LIN {X 0,Y 249.079,Z 319.46,A -85,B 0,C 180,E1 -18873.163,E2 -18873.163} C_VEL
LIN {X 0,Y 249.068,Z 319.458,A -85,B 0,C 180,E1 -18876.731,E2 -18876.731} C_VEL
LIN {X 0,Y 249.086,Z 319.447,A -85,B 0,C 180,E1 -18880.209,E2 -18880.209} C_VEL
LIN {X 0,Y 249.185,Z 319.436,A -85,B 0,C 180,E1 -18883.618,E2 -18883.618} C_VEL
LIN {X 0,Y 249.22,Z 319.439,A -85,B 0,C 180,E1 -18886.961,E2 -18886.961} C_VEL
LIN {X 0,Y 249.392,Z 319.411,A -85,B 0,C 180,E1 -18890.522,E2 -18890.522} C_VEL
LIN {X 0,Y 249.437,Z 319.395,A -85,B 0,C 180,E1 -18893.529,E2 -18893.529} C_VEL
LIN {X 0,Y 249.681,Z 319.382,A -85,B 0,C 180,E1 -18898.387,E2 -18898.387} C_VEL
LIN {X 0,Y 249.681,Z 319.38,A -85,B 0,C 180,E1 -18901.613,E2 -18901.613} C_VEL
LIN {X 0,Y 249.441,Z 319.394,A -85,B 0,C 180,E1 -18906.7,E2 -18906.7} C_VEL
LIN {X 0,Y 249.351,Z 319.418,A -85,B 0,C 180,E1 -18909.736,E2 -18909.736} C_VEL
LIN {X 0,Y 249.179,Z 319.442,A -85,B 0,C 180,E1 -18914.705,E2 -18914.705} C_VEL
LIN {X 0,Y 249.11,Z 319.452,A -85,B 0,C 180,E1 -18918.079,E2 -18918.079} C_VEL
LIN {X 0,Y 249.088,Z 319.452,A -85,B 0,C 180,E1 -18921.518,E2 -18921.518} C_VEL
LIN {X 0,Y 249.123,Z 319.451,A -85,B 0,C 180,E1 -18925.474,E2 -18925.474} C_VEL
LIN {X 0,Y 249.089,Z 319.453,A -85,B 0,C 180,E1 -18928.992,E2 -18928.992} C_VEL
LIN {X 0,Y 249.037,Z 319.46,A -85,B 0,C 180,E1 -18932.425,E2 -18932.425} C_VEL
LIN {X 0,Y 249.035,Z 319.459,A -85,B 0,C 180,E1 -18936.344,E2 -18936.344} C_VEL
LIN {X 0,Y 249.013,Z 319.458,A -85,B 0,C 180,E1 -18940.476,E2 -18940.476} C_VEL
LIN {X 0,Y 249.017,Z 319.462,A -85,B 0,C 180,E1 -18942.792,E2 -18942.792} C_VEL
LIN {X 0,Y 249.014,Z 319.464,A -85,B 0,C 180,E1 -18947.36,E2 -18947.36} C_VEL
LIN {X 0,Y 249.031,Z 319.463,A -85,B 0,C 180,E1 -18951.618,E2 -18951.618} C_VEL
LIN {X 0,Y 249.048,Z 319.46,A -85,B 0,C 180,E1 -18955.638,E2 -18955.638} C_VEL
LIN {X 0,Y 249.052,Z 319.46,A -85,B 0,C 180,E1 -18959.471,E2 -18959.471} C_VEL
LIN {X 0,Y 249.076,Z 319.457,A -85,B 0,C 180,E1 -18963.16,E2 -18963.16} C_VEL
LIN {X 0,Y 249.088,Z 319.457,A -85,B 0,C 180,E1 -18966.731,E2 -18966.731} C_VEL
LIN {X 0,Y 249.134,Z 319.449,A -85,B 0,C 180,E1 -18970.211,E2 -18970.211} C_VEL
LIN {X 0,Y 249.245,Z 319.438,A -85,B 0,C 180,E1 -18973.62,E2 -18973.62} C_VEL
LIN {X 0,Y 249.223,Z 319.441,A -85,B 0,C 180,E1 -18975.732,E2 -18975.732} C_VEL
LIN {X 0,Y 250.259,Z 322.319,A -85,B 0,C 180,E1 -18975.945,E2 -18975.945} C_VEL
LIN {X 0,Y 254.771,Z 333.047,A -85,B 0,C 180,E1 -18976.726,E2 -18976.726} C_VEL
LIN {X 0,Y 260.864,Z 350.4,A -85,B 0,C 180,E1 -18977.82,E2 -18977.82} C_VEL
LIN {X 0,Y 261.655,Z 353.279,A -85,B 0,C 180,E1 -18977.976,E2 -18977.976} C_VEL
LIN {X 0,Y 259.286,Z 425.995,A -85,B 0,C 180,E1 -18979.952,E2 -18979.952} C_VEL
LIN {X 0,Y 258.532,Z 439.131,A -85,B 0,C 180,E1 -18980.611,E2 -18980.611} C_VEL
LIN {X 0,Y 257.521,Z 451.819,A -85,B 0,C 180,E1 -18981.563,E2 -18981.563} C_VEL
LIN {X 0,Y 256.275,Z 463.159,A -85,B 0,C 180,E1 -18982.711,E2 -18982.711} C_VEL
LIN {X 0,Y 254.783,Z 475.126,A -85,B 0,C 180,E1 -18984.307,E2 -18984.307} C_VEL
LIN {X 0,Y 253.083,Z 486.09,A -85,B 0,C 180,E1 -18986.156,E2 -18986.156} C_VEL
LIN {X 0,Y 251.687,Z 494.8,A -85,B 0,C 180,E1 -18987.997,E2 -18987.997} C_VEL
LIN {X 0,Y 250.106,Z 503.926,A -85,B 0,C 180,E1 -18990.4,E2 -18990.4} C_VEL
LIN {X 0,Y 248.944,Z 511.268,A -85,B 0,C 180,E1 -18992.829,E2 -18992.829} C_VEL
LIN {X 0,Y 248.22,Z 516.233,A -85,B 0,C 180,E1 -18994.87,E2 -18994.87} C_VEL
LIN {X 0,Y 247.608,Z 521.055,A -85,B 0,C 180,E1 -18997.335,E2 -18997.335} C_VEL
LIN {X 0,Y 247.108,Z 524.766,A -85,B 0,C 180,E1 -18999.823,E2 -18999.823} C_VEL
LIN {X 0,Y 246.862,Z 526.683,A -85,B 0,C 180,E1 -19001.493,E2 -19001.493} C_VEL
LIN {X 0,Y 246.746,Z 528.928,A -85,B 0,C 180,E1 -19004.441,E2 -19004.441} C_VEL
LIN {X 0,Y 246.751,Z 529.759,A -85,B 0,C 180,E1 -19006.545,E2 -19006.545} C_VEL
LIN {X 0,Y 246.908,Z 529.939,A -85,B 0,C 180,E1 -19008.244,E2 -19008.244} C_VEL
LIN {X 0,Y 247.271,Z 529.588,A -85,B 0,C 180,E1 -19010.293,E2 -19010.293} C_VEL
LIN {X 0,Y 248.086,Z 527.931,A -85,B 0,C 180,E1 -19013.363,E2 -19013.363} C_VEL
LIN {X 0,Y 248.951,Z 525.994,A -85,B 0,C 180,E1 -19015.395,E2 -19015.395} C_VEL
LIN {X 0,Y 250.625,Z 521.798,A -85,B 0,C 180,E1 -19018.468,E2 -19018.468} C_VEL
LIN {X 0,Y 252.431,Z 516.954,A -85,B 0,C 180,E1 -19020.998,E2 -19020.998} C_VEL
LIN {X 0,Y 254.728,Z 510.734,A -85,B 0,C 180,E1 -19023.488,E2 -19023.488} C_VEL
LIN {X 0,Y 257.367,Z 502.891,A -85,B 0,C 180,E1 -19025.949,E2 -19025.949} C_VEL
LIN {X 0,Y 259.932,Z 494.763,A -85,B 0,C 180,E1 -19027.956,E2 -19027.956} C_VEL
LIN {X 0,Y 262.477,Z 485.797,A -85,B 0,C 180,E1 -19029.739,E2 -19029.739} C_VEL
LIN {X 0,Y 265.25,Z 474.762,A -85,B 0,C 180,E1 -19031.479,E2 -19031.479} C_VEL
LIN {X 0,Y 267.697,Z 463.298,A -85,B 0,C 180,E1 -19032.887,E2 -19032.887} C_VEL
LIN {X 0,Y 269.763,Z 450.842,A -85,B 0,C 180,E1 -19034.045,E2 -19034.045} C_VEL
LIN {X 0,Y 271.36,Z 438.352,A -85,B 0,C 180,E1 -19034.884,E2 -19034.884} C_VEL
LIN {X 0,Y 272.421,Z 425.844,A -85,B 0,C 180,E1 -19035.444,E2 -19035.444} C_VEL
LIN {X 0,Y 274.997,Z 366.968,A -85,B 0,C 180,E1 -19036.992,E2 -19036.992} C_VEL
LIN {X 0,Y 268.888,Z 353.819,A -85,B 0,C 180,E1 -19038.45,E2 -19038.45} C_VEL
LIN {X 0,Y 262.221,Z 341.314,A -85,B 0,C 180,E1 -19040.095,E2 -19040.095} C_VEL
LIN {X 0,Y 254.553,Z 328.6,A -85,B 0,C 180,E1 -19042.099,E2 -19042.099} C_VEL
LIN {X 0,Y 251.261,Z 323.754,A -85,B 0,C 180,E1 -19042.995,E2 -19042.995} C_VEL
LIN {X 0,Y 249.526,Z 321.295,A -85,B 0,C 180,E1 -19043.479,E2 -19043.479} C_VEL
LIN {X 0,Y 249.129,Z 320.072,A -85,B 0,C 180,E1 -19043.672,E2 -19043.672} C_VEL
LIN {X 0,Y 249.026,Z 319.443,A -85,B 0,C 180,E1 -19044.008,E2 -19044.008} C_VEL
LIN {X 0,Y 249.021,Z 319.463,A -85,B 0,C 180,E1 -19047.846,E2 -19047.846} C_VEL
LIN {X 0,Y 249.036,Z 319.458,A -85,B 0,C 180,E1 -19051.331,E2 -19051.331} C_VEL
LIN {X 0,Y 249.089,Z 319.449,A -85,B 0,C 180,E1 -19054.962,E2 -19054.962} C_VEL
LIN {X 0,Y 249.081,Z 319.448,A -85,B 0,C 180,E1 -19058.602,E2 -19058.602} C_VEL
LIN {X 0,Y 249.23,Z 319.427,A -85,B 0,C 180,E1 -19063.621,E2 -19063.621} C_VEL
LIN {X 0,Y 249.232,Z 319.427,A -85,B 0,C 180,E1 -19068.616,E2 -19068.616} C_VEL
LIN {X 0,Y 249.423,Z 319.406,A -85,B 0,C 180,E1 -19071.901,E2 -19071.901} C_VEL
LIN {X 0,Y 249.418,Z 319.409,A -85,B 0,C 180,E1 -19076.77,E2 -19076.77} C_VEL
LIN {X 0,Y 249.715,Z 319.375,A -85,B 0,C 180,E1 -19080,E2 -19080} C_VEL
LIN {X 0,Y 249.421,Z 319.397,A -85,B 0,C 180,E1 -19083.231,E2 -19083.231} C_VEL
LIN {X 0,Y 249.447,Z 319.398,A -85,B 0,C 180,E1 -19087.739,E2 -19087.739} C_VEL
LIN {X 0,Y 248.791,Z 319.482,A -85,B 0,C 180,E1 -19089.084,E2 -19089.084} C_VEL
LIN {X 0,Y 245.807,Z 319.865,A -85,B 0,C 180,E1 -19091.272,E2 -19091.272} C_VEL
LIN {X 0,Y 243.266,Z 320.171,A -85,B 0,C 180,E1 -19093.055,E2 -19093.055} C_VEL
LIN {X 0,Y 242.208,Z 320.299,A -85,B 0,C 180,E1 -19094.443,E2 -19094.443} C_VEL
LIN {X 0,Y 242.142,Z 320.311,A -85,B 0,C 180,E1 -19094.913,E2 -19094.913} C_VEL
LIN {X 0,Y 242.062,Z 320.318,A -85,B 0,C 180,E1 -19098.625,E2 -19098.625} C_VEL
LIN {X 0,Y 242.002,Z 320.336,A -85,B 0,C 180,E1 -19102.181,E2 -19102.181} C_VEL
LIN {X 0,Y 242.056,Z 320.334,A -85,B 0,C 180,E1 -19105.84,E2 -19105.84} C_VEL
LIN {X 0,Y 242.021,Z 320.335,A -85,B 0,C 180,E1 -19109.582,E2 -19109.582} C_VEL
LIN {X 0,Y 241.982,Z 320.341,A -85,B 0,C 180,E1 -19113.493,E2 -19113.493} C_VEL
LIN {X 0,Y 242.005,Z 320.345,A -85,B 0,C 180,E1 -19117.58,E2 -19117.58} C_VEL
LIN {X 0,Y 241.962,Z 320.342,A -85,B 0,C 180,E1 -19121.918,E2 -19121.918} C_VEL
LIN {X 0,Y 241.956,Z 320.354,A -85,B 0,C 180,E1 -19123.861,E2 -19123.861} C_VEL
LIN {X 0,Y 244.234,Z 327.54,A -85,B 0,C 180,E1 -19127.815,E2 -19127.815} C_VEL
LIN {X 0,Y 245.915,Z 333.614,A -85,B 0,C 180,E1 -19130.733,E2 -19130.733} C_VEL
LIN {X 0,Y 248.478,Z 338.048,A -85,B 0,C 180,E1 -19131.493,E2 -19131.493} C_VEL
LIN {X 0,Y 254.393,Z 348.559,A -85,B 0,C 180,E1 -19133.168,E2 -19133.168} C_VEL
LIN {X 0,Y 260.731,Z 361.176,A -85,B 0,C 180,E1 -19134.877,E2 -19134.877} C_VEL
LIN {X 0,Y 265.439,Z 371.761,A -85,B 0,C 180,E1 -19136.103,E2 -19136.103} C_VEL
LIN {X 0,Y 268.42,Z 390.693,A -85,B 0,C 180,E1 -19137.259,E2 -19137.259} C_VEL
LIN {X 0,Y 265.995,Z 443.364,A -85,B 0,C 180,E1 -19138.684,E2 -19138.684} C_VEL
LIN {X 0,Y 264.584,Z 457.091,A -85,B 0,C 180,E1 -19139.33,E2 -19139.33} C_VEL
LIN {X 0,Y 262.579,Z 469.788,A -85,B 0,C 180,E1 -19140.213,E2 -19140.213} C_VEL
LIN {X 0,Y 260.163,Z 481.585,A -85,B 0,C 180,E1 -19141.351,E2 -19141.351} C_VEL
LIN {X 0,Y 257.684,Z 491.661,A -85,B 0,C 180,E1 -19142.6,E2 -19142.6} C_VEL
LIN {X 0,Y 254.822,Z 502.14,A -85,B 0,C 180,E1 -19144.257,E2 -19144.257} C_VEL
LIN {X 0,Y 251.917,Z 511.618,A -85,B 0,C 180,E1 -19146.142,E2 -19146.142} C_VEL
LIN {X 0,Y 248.731,Z 520.781,A -85,B 0,C 180,E1 -19148.452,E2 -19148.452} C_VEL
LIN {X 0,Y 246.35,Z 528.171,A -85,B 0,C 180,E1 -19150.851,E2 -19150.851} C_VEL
LIN {X 0,Y 244.26,Z 534.136,A -85,B 0,C 180,E1 -19153.281,E2 -19153.281} C_VEL
LIN {X 0,Y 242.422,Z 538.878,A -85,B 0,C 180,E1 -19155.737,E2 -19155.737} C_VEL
LIN {X 0,Y 241.211,Z 542.533,A -85,B 0,C 180,E1 -19158.234,E2 -19158.234} C_VEL
LIN {X 0,Y 240.639,Z 544.439,A -85,B 0,C 180,E1 -19159.91,E2 -19159.91} C_VEL
LIN {X 0,Y 240.214,Z 545.898,A -85,B 0,C 180,E1 -19161.591,E2 -19161.591} C_VEL
LIN {X 0,Y 239.841,Z 547.621,A -85,B 0,C 180,E1 -19164.959,E2 -19164.959} C_VEL
LIN {X 0,Y 239.82,Z 547.911,A -85,B 0,C 180,E1 -19166.642,E2 -19166.642} C_VEL
LIN {X 0,Y 239.903,Z 547.793,A -85,B 0,C 180,E1 -19168.324,E2 -19168.324} C_VEL
LIN {X 0,Y 239.958,Z 547.253,A -85,B 0,C 180,E1 -19170.003,E2 -19170.003} C_VEL
LIN {X 0,Y 239.953,Z 546.315,A -85,B 0,C 180,E1 -19171.681,E2 -19171.681} C_VEL
LIN {X 0,Y 239.892,Z 544.97,A -85,B 0,C 180,E1 -19173.362,E2 -19173.362} C_VEL
LIN {X 0,Y 239.922,Z 542.099,A -85,B 0,C 180,E1 -19175.886,E2 -19175.886} C_VEL
LIN {X 0,Y 240.201,Z 538.173,A -85,B 0,C 180,E1 -19178.415,E2 -19178.415} C_VEL
LIN {X 0,Y 240.827,Z 532.102,A -85,B 0,C 180,E1 -19181.363,E2 -19181.363} C_VEL
LIN {X 0,Y 241.786,Z 525.416,A -85,B 0,C 180,E1 -19183.877,E2 -19183.877} C_VEL
LIN {X 0,Y 243.16,Z 517.097,A -85,B 0,C 180,E1 -19186.37,E2 -19186.37} C_VEL
LIN {X 0,Y 244.587,Z 508.167,A -85,B 0,C 180,E1 -19188.516,E2 -19188.516} C_VEL
LIN {X 0,Y 246.257,Z 497.98,A -85,B 0,C 180,E1 -19190.466,E2 -19190.466} C_VEL
LIN {X 0,Y 247.77,Z 487.482,A -85,B 0,C 180,E1 -19192.078,E2 -19192.078} C_VEL
LIN {X 0,Y 249.502,Z 476.011,A -85,B 0,C 180,E1 -19193.448,E2 -19193.448} C_VEL
LIN {X 0,Y 250.861,Z 464.137,A -85,B 0,C 180,E1 -19194.52,E2 -19194.52} C_VEL
LIN {X 0,Y 251.995,Z 451.358,A -85,B 0,C 180,E1 -19195.338,E2 -19195.338} C_VEL
LIN {X 0,Y 252.7,Z 438.181,A -85,B 0,C 180,E1 -19195.87,E2 -19195.87} C_VEL
LIN {X 0,Y 254.188,Z 385.832,A -85,B 0,C 180,E1 -19197.324,E2 -19197.324} C_VEL
LIN {X 0,Y 249.433,Z 347.285,A -85,B 0,C 180,E1 -19198.962,E2 -19198.962} C_VEL
LIN {X 0,Y 245.183,Z 335.103,A -85,B 0,C 180,E1 -19199.805,E2 -19199.805} C_VEL
LIN {X 0,Y 242.879,Z 324.284,A -85,B 0,C 180,E1 -19203.853,E2 -19203.853} C_VEL
LIN {X 0,Y 242.016,Z 320.338,A -85,B 0,C 180,E1 -19205.445,E2 -19205.445} C_VEL
LIN {X 0,Y 241.963,Z 320.345,A -85,B 0,C 180,E1 -19209.72,E2 -19209.72} C_VEL
LIN {X 0,Y 241.926,Z 320.349,A -85,B 0,C 180,E1 -19214.206,E2 -19214.206} C_VEL
LIN {X 0,Y 241.941,Z 320.346,A -85,B 0,C 180,E1 -19218.078,E2 -19218.078} C_VEL
LIN {X 0,Y 241.994,Z 320.338,A -85,B 0,C 180,E1 -19222.418,E2 -19222.418} C_VEL
LIN {X 0,Y 241.988,Z 320.337,A -85,B 0,C 180,E1 -19226.508,E2 -19226.508} C_VEL
LIN {X 0,Y 242.045,Z 320.329,A -85,B 0,C 180,E1 -19230.588,E2 -19230.588} C_VEL
LIN {X 0,Y 242.076,Z 320.329,A -85,B 0,C 180,E1 -19234.184,E2 -19234.184} C_VEL
LIN {X 0,Y 242.031,Z 320.333,A -85,B 0,C 180,E1 -19238.316,E2 -19238.316} C_VEL
LIN {X 0,Y 242.124,Z 320.312,A -85,B 0,C 180,E1 -19243.316,E2 -19243.316} C_VEL
LIN {X 0,Y 242.186,Z 320.314,A -85,B 0,C 180,E1 -19248.279,E2 -19248.279} C_VEL
LIN {X 0,Y 242.38,Z 320.279,A -85,B 0,C 180,E1 -19251.664,E2 -19251.664} C_VEL
LIN {X 0,Y 242.249,Z 320.295,A -85,B 0,C 180,E1 -19255.007,E2 -19255.007} C_VEL
LIN {X 0,Y 242.642,Z 320.259,A -85,B 0,C 180,E1 -19258.34,E2 -19258.34} C_VEL
LIN {X 0,Y 242.642,Z 320.257,A -85,B 0,C 180,E1 -19261.659,E2 -19261.659} C_VEL
LIN {X 0,Y 242.423,Z 320.268,A -85,B 0,C 180,E1 -19266.672,E2 -19266.672} C_VEL
LIN {X 0,Y 242.275,Z 320.3,A -85,B 0,C 180,E1 -19270.023,E2 -19270.023} C_VEL
LIN {X 0,Y 242.134,Z 320.317,A -85,B 0,C 180,E1 -19275.143,E2 -19275.143} C_VEL
LIN {X 0,Y 242.049,Z 320.335,A -85,B 0,C 180,E1 -19278.626,E2 -19278.626} C_VEL
LIN {X 0,Y 242.011,Z 320.333,A -85,B 0,C 180,E1 -19282.18,E2 -19282.18} C_VEL
LIN {X 0,Y 242.074,Z 320.328,A -85,B 0,C 180,E1 -19285.837,E2 -19285.837} C_VEL
LIN {X 0,Y 242.037,Z 320.331,A -85,B 0,C 180,E1 -19289.579,E2 -19289.579} C_VEL
LIN {X 0,Y 241.987,Z 320.337,A -85,B 0,C 180,E1 -19293.491,E2 -19293.491} C_VEL
LIN {X 0,Y 241.993,Z 320.339,A -85,B 0,C 180,E1 -19297.581,E2 -19297.581} C_VEL
LIN {X 0,Y 241.945,Z 320.344,A -85,B 0,C 180,E1 -19301.92,E2 -19301.92} C_VEL
LIN {X 0,Y 241.932,Z 320.344,A -85,B 0,C 180,E1 -19306.571,E2 -19306.571} C_VEL
LIN {X 0,Y 241.961,Z 320.341,A -85,B 0,C 180,E1 -19310.279,E2 -19310.279} C_VEL
LIN {X 0,Y 241.993,Z 320.338,A -85,B 0,C 180,E1 -19314.488,E2 -19314.488} C_VEL
LIN {X 0,Y 241.977,Z 320.341,A -85,B 0,C 180,E1 -19318.478,E2 -19318.478} C_VEL
LIN {X 0,Y 242.007,Z 320.339,A -85,B 0,C 180,E1 -19322.31,E2 -19322.31} C_VEL
LIN {X 0,Y 242.064,Z 320.333,A -85,B 0,C 180,E1 -19326.014,E2 -19326.014} C_VEL
LIN {X 0,Y 242.064,Z 320.329,A -85,B 0,C 180,E1 -19329.608,E2 -19329.608} C_VEL
LIN {X 0,Y 242.166,Z 320.32,A -85,B 0,C 180,E1 -19333.276,E2 -19333.276} C_VEL
LIN {X 0,Y 242.169,Z 320.318,A -85,B 0,C 180,E1 -19334.988,E2 -19334.988} C_VEL
LIN {X 0,Y 243.233,Z 323.279,A -85,B 0,C 180,E1 -19335.234,E2 -19335.234} C_VEL
LIN {X 0,Y 247.549,Z 332.958,A -85,B 0,C 180,E1 -19336,E2 -19336} C_VEL
LIN {X 0,Y 254.442,Z 352.277,A -85,B 0,C 180,E1 -19337.282,E2 -19337.282} C_VEL
LIN {X 0,Y 255.026,Z 354.157,A -85,B 0,C 180,E1 -19337.394,E2 -19337.394} C_VEL
LIN {X 0,Y 252.608,Z 426.79,A -85,B 0,C 180,E1 -19339.427,E2 -19339.427} C_VEL
LIN {X 0,Y 251.761,Z 440.555,A -85,B 0,C 180,E1 -19340.153,E2 -19340.153} C_VEL
LIN {X 0,Y 250.737,Z 452.917,A -85,B 0,C 180,E1 -19341.13,E2 -19341.13} C_VEL
LIN {X 0,Y 249.425,Z 464.032,A -85,B 0,C 180,E1 -19342.306,E2 -19342.306} C_VEL
LIN {X 0,Y 248.065,Z 474.734,A -85,B 0,C 180,E1 -19343.767,E2 -19343.767} C_VEL
LIN {X 0,Y 246.256,Z 486.013,A -85,B 0,C 180,E1 -19345.701,E2 -19345.701} C_VEL
LIN {X 0,Y 244.832,Z 494.536,A -85,B 0,C 180,E1 -19347.53,E2 -19347.53} C_VEL
LIN {X 0,Y 243.197,Z 503.765,A -85,B 0,C 180,E1 -19349.998,E2 -19349.998} C_VEL
LIN {X 0,Y 241.966,Z 511.183,A -85,B 0,C 180,E1 -19352.495,E2 -19352.495} C_VEL
LIN {X 0,Y 241.093,Z 517.128,A -85,B 0,C 180,E1 -19355.014,E2 -19355.014} C_VEL
LIN {X 0,Y 240.473,Z 521.82,A -85,B 0,C 180,E1 -19357.554,E2 -19357.554} C_VEL
LIN {X 0,Y 239.953,Z 525.411,A -85,B 0,C 180,E1 -19360.119,E2 -19360.119} C_VEL
LIN {X 0,Y 239.75,Z 527.213,A -85,B 0,C 180,E1 -19361.838,E2 -19361.838} C_VEL
LIN {X 0,Y 239.655,Z 529.203,A -85,B 0,C 180,E1 -19364.594,E2 -19364.594} C_VEL
LIN {X 0,Y 239.684,Z 530.09,A -85,B 0,C 180,E1 -19367.048,E2 -19367.048} C_VEL
LIN {X 0,Y 239.893,Z 530.183,A -85,B 0,C 180,E1 -19368.797,E2 -19368.797} C_VEL
LIN {X 0,Y 240.24,Z 529.86,A -85,B 0,C 180,E1 -19370.589,E2 -19370.589} C_VEL
LIN {X 0,Y 240.656,Z 529.148,A -85,B 0,C 180,E1 -19372.309,E2 -19372.309} C_VEL
LIN {X 0,Y 241.257,Z 527.942,A -85,B 0,C 180,E1 -19374.066,E2 -19374.066} C_VEL
LIN {X 0,Y 242.475,Z 525.304,A -85,B 0,C 180,E1 -19376.692,E2 -19376.692} C_VEL
LIN {X 0,Y 244.055,Z 521.552,A -85,B 0,C 180,E1 -19379.308,E2 -19379.308} C_VEL
LIN {X 0,Y 246.032,Z 516.566,A -85,B 0,C 180,E1 -19381.898,E2 -19381.898} C_VEL
LIN {X 0,Y 248.51,Z 510.192,A -85,B 0,C 180,E1 -19384.441,E2 -19384.441} C_VEL
LIN {X 0,Y 251.388,Z 502.122,A -85,B 0,C 180,E1 -19386.943,E2 -19386.943} C_VEL
LIN {X 0,Y 254.274,Z 493.012,A -85,B 0,C 180,E1 -19389.158,E2 -19389.158} C_VEL
LIN {X 0,Y 257.105,Z 483.439,A -85,B 0,C 180,E1 -19390.995,E2 -19390.995} C_VEL
LIN {X 0,Y 259.708,Z 473.148,A -85,B 0,C 180,E1 -19392.569,E2 -19392.569} C_VEL
LIN {X 0,Y 262.245,Z 461.061,A -85,B 0,C 180,E1 -19394.002,E2 -19394.002} C_VEL
LIN {X 0,Y 264.216,Z 449.064,A -85,B 0,C 180,E1 -19395.086,E2 -19395.086} C_VEL
LIN {X 0,Y 265.774,Z 436.705,A -85,B 0,C 180,E1 -19395.877,E2 -19395.877} C_VEL
LIN {X 0,Y 266.835,Z 424.087,A -85,B 0,C 180,E1 -19396.394,E2 -19396.394} C_VEL
LIN {X 0,Y 269.338,Z 369.122,A -85,B 0,C 180,E1 -19397.852,E2 -19397.852} C_VEL
LIN {X 0,Y 263.234,Z 356.083,A -85,B 0,C 180,E1 -19399.377,E2 -19399.377} C_VEL
LIN {X 0,Y 255.57,Z 342.012,A -85,B 0,C 180,E1 -19401.376,E2 -19401.376} C_VEL
LIN {X 0,Y 249.809,Z 332.638,A -85,B 0,C 180,E1 -19402.962,E2 -19402.962} C_VEL
LIN {X 0,Y 247.435,Z 329.138,A -85,B 0,C 180,E1 -19403.636,E2 -19403.636} C_VEL
LIN {X 0,Y 245.35,Z 326.004,A -85,B 0,C 180,E1 -19404.247,E2 -19404.247} C_VEL
LIN {X 0,Y 244.417,Z 324.846,A -85,B 0,C 180,E1 -19404.516,E2 -19404.516} C_VEL
LIN {X 0,Y 242.517,Z 322.265,A -85,B 0,C 180,E1 -19405.087,E2 -19405.087} C_VEL
LIN {X 0,Y 242.018,Z 320.518,A -85,B 0,C 180,E1 -19405.321,E2 -19405.321} C_VEL
LIN {X 0,Y 241.94,Z 320.342,A -85,B 0,C 180,E1 -19408.475,E2 -19408.475} C_VEL
LIN {X 0,Y 241.955,Z 320.34,A -85,B 0,C 180,E1 -19412.307,E2 -19412.307} C_VEL
LIN {X 0,Y 242.013,Z 320.332,A -85,B 0,C 180,E1 -19416.012,E2 -19416.012} C_VEL
LIN {X 0,Y 242.023,Z 320.326,A -85,B 0,C 180,E1 -19419.607,E2 -19419.607} C_VEL
LIN {X 0,Y 242.151,Z 320.308,A -85,B 0,C 180,E1 -19423.278,E2 -19423.278} C_VEL
LIN {X 0,Y 242.168,Z 320.305,A -85,B 0,C 180,E1 -19428.279,E2 -19428.279} C_VEL
LIN {X 0,Y 242.373,Z 320.286,A -85,B 0,C 180,E1 -19431.664,E2 -19431.664} C_VEL
LIN {X 0,Y 242.233,Z 320.31,A -85,B 0,C 180,E1 -19435.007,E2 -19435.007} C_VEL
LIN {X 0,Y 242.622,Z 320.246,A -85,B 0,C 180,E1 -19438.34,E2 -19438.34} C_VEL
LIN {X 0,Y 242.623,Z 320.258,A -85,B 0,C 180,E1 -19441.66,E2 -19441.66} C_VEL
LIN {X 0,Y 242.394,Z 320.276,A -85,B 0,C 180,E1 -19447.745,E2 -19447.745} C_VEL
LIN {X 0,Y 242.302,Z 320.295,A -85,B 0,C 180,E1 -19450.023,E2 -19450.023} C_VEL
LIN {X 0,Y 242.142,Z 320.311,A -85,B 0,C 180,E1 -19454.913,E2 -19454.913} C_VEL
LIN {X 0,Y 241.521,Z 320.402,A -85,B 0,C 180,E1 -19456.3,E2 -19456.3} C_VEL
LIN {X 0,Y 238.655,Z 320.771,A -85,B 0,C 180,E1 -19458.561,E2 -19458.561} C_VEL
LIN {X 0,Y 236.167,Z 321.077,A -85,B 0,C 180,E1 -19460.403,E2 -19460.403} C_VEL
LIN {X 0,Y 235.069,Z 321.203,A -85,B 0,C 180,E1 -19461.834,E2 -19461.834} C_VEL
LIN {X 0,Y 234.965,Z 321.21,A -85,B 0,C 180,E1 -19462.319,E2 -19462.319} C_VEL
LIN {X 0,Y 234.96,Z 321.213,A -85,B 0,C 180,E1 -19466.659,E2 -19466.659} C_VEL
LIN {X 0,Y 234.923,Z 321.223,A -85,B 0,C 180,E1 -19470.569,E2 -19470.569} C_VEL
LIN {X 0,Y 234.952,Z 321.219,A -85,B 0,C 180,E1 -19474.635,E2 -19474.635} C_VEL
LIN {X 0,Y 234.959,Z 321.214,A -85,B 0,C 180,E1 -19478.954,E2 -19478.954} C_VEL
LIN {X 0,Y 234.927,Z 321.303,A -85,B 0,C 180,E1 -19482.328,E2 -19482.328} C_VEL
LIN {X 0,Y 237.543,Z 329.57,A -85,B 0,C 180,E1 -19487.123,E2 -19487.123} C_VEL
LIN {X 0,Y 238.558,Z 333.073,A -85,B 0,C 180,E1 -19488.923,E2 -19488.923} C_VEL
LIN {X 0,Y 241.281,Z 337.753,A -85,B 0,C 180,E1 -19489.806,E2 -19489.806} C_VEL
LIN {X 0,Y 247.872,Z 349.115,A -85,B 0,C 180,E1 -19491.802,E2 -19491.802} C_VEL
LIN {X 0,Y 254.514,Z 362.104,A -85,B 0,C 180,E1 -19493.704,E2 -19493.704} C_VEL
LIN {X 0,Y 260.214,Z 374.792,A -85,B 0,C 180,E1 -19495.271,E2 -19495.271} C_VEL
LIN {X 0,Y 262.808,Z 391.644,A -85,B 0,C 180,E1 -19496.334,E2 -19496.334} C_VEL
LIN {X 0,Y 260.27,Z 443.79,A -85,B 0,C 180,E1 -19497.774,E2 -19497.774} C_VEL
LIN {X 0,Y 258.813,Z 457.288,A -85,B 0,C 180,E1 -19498.431,E2 -19498.431} C_VEL
LIN {X 0,Y 256.703,Z 470.054,A -85,B 0,C 180,E1 -19499.345,E2 -19499.345} C_VEL
LIN {X 0,Y 254.35,Z 480.952,A -85,B 0,C 180,E1 -19500.405,E2 -19500.405} C_VEL
LIN {X 0,Y 251.441,Z 492.375,A -85,B 0,C 180,E1 -19501.86,E2 -19501.86} C_VEL
LIN {X 0,Y 248.472,Z 502.688,A -85,B 0,C 180,E1 -19503.549,E2 -19503.549} C_VEL
LIN {X 0,Y 245.469,Z 511.998,A -85,B 0,C 180,E1 -19505.474,E2 -19505.474} C_VEL
LIN {X 0,Y 242.164,Z 521.026,A -85,B 0,C 180,E1 -19507.838,E2 -19507.838} C_VEL
LIN {X 0,Y 239.641,Z 528.321,A -85,B 0,C 180,E1 -19510.293,E2 -19510.293} C_VEL
LIN {X 0,Y 237.459,Z 534.203,A -85,B 0,C 180,E1 -19512.787,E2 -19512.787} C_VEL
LIN {X 0,Y 235.524,Z 538.872,A -85,B 0,C 180,E1 -19515.31,E2 -19515.31} C_VEL
LIN {X 0,Y 234.247,Z 542.46,A -85,B 0,C 180,E1 -19517.879,E2 -19517.879} C_VEL
LIN {X 0,Y 233.613,Z 544.322,A -85,B 0,C 180,E1 -19519.604,E2 -19519.604} C_VEL
LIN {X 0,Y 232.889,Z 546.757,A -85,B 0,C 180,E1 -19523.07,E2 -19523.07} C_VEL
LIN {X 0,Y 232.761,Z 547.495,A -85,B 0,C 180,E1 -19525.145,E2 -19525.145} C_VEL
LIN {X 0,Y 232.811,Z 547.484,A -85,B 0,C 180,E1 -19528.273,E2 -19528.273} C_VEL
LIN {X 0,Y 232.888,Z 546.915,A -85,B 0,C 180,E1 -19530.003,E2 -19530.003} C_VEL
LIN {X 0,Y 232.86,Z 545.947,A -85,B 0,C 180,E1 -19531.732,E2 -19531.732} C_VEL
LIN {X 0,Y 232.795,Z 544.568,A -85,B 0,C 180,E1 -19533.464,E2 -19533.464} C_VEL
LIN {X 0,Y 232.843,Z 541.637,A -85,B 0,C 180,E1 -19536.067,E2 -19536.067} C_VEL
LIN {X 0,Y 233.137,Z 537.644,A -85,B 0,C 180,E1 -19538.672,E2 -19538.672} C_VEL
LIN {X 0,Y 233.817,Z 531.463,A -85,B 0,C 180,E1 -19541.708,E2 -19541.708} C_VEL
LIN {X 0,Y 234.876,Z 524.697,A -85,B 0,C 180,E1 -19544.294,E2 -19544.294} C_VEL
LIN {X 0,Y 236.335,Z 516.282,A -85,B 0,C 180,E1 -19546.857,E2 -19546.857} C_VEL
LIN {X 0,Y 237.745,Z 507.578,A -85,B 0,C 180,E1 -19548.978,E2 -19548.978} C_VEL
LIN {X 0,Y 239.37,Z 498.034,A -85,B 0,C 180,E1 -19550.857,E2 -19550.857} C_VEL
LIN {X 0,Y 240.923,Z 487.601,A -85,B 0,C 180,E1 -19552.514,E2 -19552.514} C_VEL
LIN {X 0,Y 242.707,Z 476.224,A -85,B 0,C 180,E1 -19553.918,E2 -19553.918} C_VEL
LIN {X 0,Y 244.111,Z 464.569,A -85,B 0,C 180,E1 -19555.017,E2 -19555.017} C_VEL
LIN {X 0,Y 245.349,Z 451.155,A -85,B 0,C 180,E1 -19555.905,E2 -19555.905} C_VEL
LIN {X 0,Y 246.075,Z 438.014,A -85,B 0,C 180,E1 -19556.449,E2 -19556.449} C_VEL
LIN {X 0,Y 247.614,Z 386.608,A -85,B 0,C 180,E1 -19557.911,E2 -19557.911} C_VEL
LIN {X 0,Y 243.017,Z 349.091,A -85,B 0,C 180,E1 -19559.559,E2 -19559.559} C_VEL
LIN {X 0,Y 237.857,Z 334.84,A -85,B 0,C 180,E1 -19560.599,E2 -19560.599} C_VEL
LIN {X 0,Y 235.745,Z 324.785,A -85,B 0,C 180,E1 -19564.504,E2 -19564.504} C_VEL
LIN {X 0,Y 234.968,Z 321.214,A -85,B 0,C 180,E1 -19565.98,E2 -19565.98} C_VEL
LIN {X 0,Y 234.949,Z 321.22,A -85,B 0,C 180,E1 -19568.946,E2 -19568.946} C_VEL
LIN {X 0,Y 234.886,Z 321.226,A -85,B 0,C 180,E1 -19573.489,E2 -19573.489} C_VEL
LIN {X 0,Y 234.886,Z 321.226,A -85,B 0,C 180,E1 -19576.513,E2 -19576.513} C_VEL
LIN {X 0,Y 234.926,Z 321.22,A -85,B 0,C 180,E1 -19581.08,E2 -19581.08} C_VEL
LIN {X 0,Y 234.935,Z 321.216,A -85,B 0,C 180,E1 -19585.362,E2 -19585.362} C_VEL
LIN {X 0,Y 234.94,Z 321.215,A -85,B 0,C 180,E1 -19589.433,E2 -19589.433} C_VEL
LIN {X 0,Y 235.003,Z 321.211,A -85,B 0,C 180,E1 -19593.794,E2 -19593.794} C_VEL
LIN {X 0,Y 234.996,Z 321.21,A -85,B 0,C 180,E1 -19598.968,E2 -19598.968} C_VEL
LIN {X 0,Y 235.064,Z 321.189,A -85,B 0,C 180,E1 -19603.092,E2 -19603.092} C_VEL
LIN {X 0,Y 235.118,Z 321.197,A -85,B 0,C 180,E1 -19607.922,E2 -19607.922} C_VEL
LIN {X 0,Y 235.319,Z 321.16,A -85,B 0,C 180,E1 -19611.412,E2 -19611.412} C_VEL
LIN {X 0,Y 235.358,Z 321.146,A -85,B 0,C 180,E1 -19613.14,E2 -19613.14} C_VEL
LIN {X 0,Y 235.601,Z 321.137,A -85,B 0,C 180,E1 -19618.29,E2 -19618.29} C_VEL
LIN {X 0,Y 235.602,Z 321.134,A -85,B 0,C 180,E1 -19621.709,E2 -19621.709} C_VEL
LIN {X 0,Y 235.374,Z 321.146,A -85,B 0,C 180,E1 -19626.859,E2 -19626.859} C_VEL
LIN {X 0,Y 235.221,Z 321.181,A -85,B 0,C 180,E1 -19630.327,E2 -19630.327} C_VEL
LIN {X 0,Y 235.081,Z 321.194,A -85,B 0,C 180,E1 -19635.608,E2 -19635.608} C_VEL
LIN {X 0,Y 234.991,Z 321.212,A -85,B 0,C 180,E1 -19639.207,E2 -19639.207} C_VEL
LIN {X 0,Y 234.958,Z 321.213,A -85,B 0,C 180,E1 -19642.883,E2 -19642.883} C_VEL
LIN {X 0,Y 234.976,Z 321.215,A -85,B 0,C 180,E1 -19646.656,E2 -19646.656} C_VEL
LIN {X 0,Y 234.938,Z 321.215,A -85,B 0,C 180,E1 -19650.566,E2 -19650.566} C_VEL
LIN {X 0,Y 234.933,Z 321.214,A -85,B 0,C 180,E1 -19654.637,E2 -19654.637} C_VEL
LIN {X 0,Y 234.948,Z 321.216,A -85,B 0,C 180,E1 -19658.943,E2 -19658.943} C_VEL
LIN {X 0,Y 234.892,Z 321.225,A -85,B 0,C 180,E1 -19663.484,E2 -19663.484} C_VEL
LIN {X 0,Y 234.885,Z 321.222,A -85,B 0,C 180,E1 -19666.511,E2 -19666.511} C_VEL
LIN {X 0,Y 234.923,Z 321.217,A -85,B 0,C 180,E1 -19671.077,E2 -19671.077} C_VEL
LIN {X 0,Y 234.935,Z 321.217,A -85,B 0,C 180,E1 -19675.36,E2 -19675.36} C_VEL
LIN {X 0,Y 234.926,Z 321.219,A -85,B 0,C 180,E1 -19679.429,E2 -19679.429} C_VEL
LIN {X 0,Y 234.997,Z 321.213,A -85,B 0,C 180,E1 -19683.792,E2 -19683.792} C_VEL
LIN {X 0,Y 235.031,Z 321.205,A -85,B 0,C 180,E1 -19688.969,E2 -19688.969} C_VEL
LIN {X 0,Y 235.115,Z 321.199,A -85,B 0,C 180,E1 -19694.225,E2 -19694.225} C_VEL
LIN {X 0,Y 236.2,Z 324.171,A -85,B 0,C 180,E1 -19694.477,E2 -19694.477} C_VEL
LIN {X 0,Y 241.344,Z 335.447,A -85,B 0,C 180,E1 -19695.424,E2 -19695.424} C_VEL
LIN {X 0,Y 247.993,Z 354.095,A -85,B 0,C 180,E1 -19696.709,E2 -19696.709} C_VEL
LIN {X 0,Y 248.457,Z 355.643,A -85,B 0,C 180,E1 -19696.804,E2 -19696.804} C_VEL
LIN {X 0,Y 246.013,Z 426.517,A -85,B 0,C 180,E1 -19698.827,E2 -19698.827} C_VEL
LIN {X 0,Y 245.175,Z 439.709,A -85,B 0,C 180,E1 -19699.52,E2 -19699.52} C_VEL
LIN {X 0,Y 244.054,Z 452.929,A -85,B 0,C 180,E1 -19700.571,E2 -19700.571} C_VEL
LIN {X 0,Y 242.591,Z 464.9,A -85,B 0,C 180,E1 -19701.878,E2 -19701.878} C_VEL
LIN {X 0,Y 241.017,Z 476.53,A -85,B 0,C 180,E1 -19703.542,E2 -19703.542} C_VEL
LIN {X 0,Y 239.32,Z 486.682,A -85,B 0,C 180,E1 -19705.365,E2 -19705.365} C_VEL
LIN {X 0,Y 237.724,Z 495.951,A -85,B 0,C 180,E1 -19707.456,E2 -19707.456} C_VEL
LIN {X 0,Y 236.061,Z 504.971,A -85,B 0,C 180,E1 -19709.997,E2 -19709.997} C_VEL
LIN {X 0,Y 234.827,Z 512.222,A -85,B 0,C 180,E1 -19712.57,E2 -19712.57} C_VEL
LIN {X 0,Y 233.964,Z 517.993,A -85,B 0,C 180,E1 -19715.168,E2 -19715.168} C_VEL
LIN {X 0,Y 233.327,Z 522.545,A -85,B 0,C 180,E1 -19717.787,E2 -19717.787} C_VEL
LIN {X 0,Y 232.823,Z 526.014,A -85,B 0,C 180,E1 -19720.432,E2 -19720.432} C_VEL
LIN {X 0,Y 232.621,Z 527.74,A -85,B 0,C 180,E1 -19722.207,E2 -19722.207} C_VEL
LIN {X 0,Y 232.575,Z 529.482,A -85,B 0,C 180,E1 -19724.765,E2 -19724.765} C_VEL
LIN {X 0,Y 232.64,Z 530.391,A -85,B 0,C 180,E1 -19727.581,E2 -19727.581} C_VEL
LIN {X 0,Y 233.202,Z 530.135,A -85,B 0,C 180,E1 -19730.894,E2 -19730.894} C_VEL
LIN {X 0,Y 233.772,Z 529.227,A -85,B 0,C 180,E1 -19733.003,E2 -19733.003} C_VEL
LIN {X 0,Y 235.168,Z 526.571,A -85,B 0,C 180,E1 -19736.292,E2 -19736.292} C_VEL
LIN {X 0,Y 236.895,Z 522.757,A -85,B 0,C 180,E1 -19739.305,E2 -19739.305} C_VEL
LIN {X 0,Y 238.917,Z 518.066,A -85,B 0,C 180,E1 -19741.967,E2 -19741.967} C_VEL
LIN {X 0,Y 241.411,Z 511.992,A -85,B 0,C 180,E1 -19744.586,E2 -19744.586} C_VEL
LIN {X 0,Y 244.321,Z 504.315,A -85,B 0,C 180,E1 -19747.159,E2 -19747.159} C_VEL
LIN {X 0,Y 247.006,Z 496.663,A -85,B 0,C 180,E1 -19749.194,E2 -19749.194} C_VEL
LIN {X 0,Y 249.835,Z 487.749,A -85,B 0,C 180,E1 -19751.11,E2 -19751.11} C_VEL
LIN {X 0,Y 252.851,Z 477.041,A -85,B 0,C 180,E1 -19752.916,E2 -19752.916} C_VEL
LIN {X 0,Y 255.627,Z 465.327,A -85,B 0,C 180,E1 -19754.456,E2 -19754.456} C_VEL
LIN {X 0,Y 257.867,Z 453.25,A -85,B 0,C 180,E1 -19755.674,E2 -19755.674} C_VEL
LIN {X 0,Y 259.689,Z 440.592,A -85,B 0,C 180,E1 -19756.588,E2 -19756.588} C_VEL
LIN {X 0,Y 260.985,Z 427.501,A -85,B 0,C 180,E1 -19757.22,E2 -19757.22} C_VEL
LIN {X 0,Y 263.683,Z 371.271,A -85,B 0,C 180,E1 -19758.76,E2 -19758.76} C_VEL
LIN {X 0,Y 258.193,Z 359.618,A -85,B 0,C 180,E1 -19760.2,E2 -19760.2} C_VEL
LIN {X 0,Y 251.176,Z 346.522,A -85,B 0,C 180,E1 -19762.119,E2 -19762.119} C_VEL
LIN {X 0,Y 245.724,Z 337.561,A -85,B 0,C 180,E1 -19763.684,E2 -19763.684} C_VEL
LIN {X 0,Y 240.701,Z 330.266,A -85,B 0,C 180,E1 -19765.195,E2 -19765.195} C_VEL
LIN {X 0,Y 238.508,Z 327.052,A -85,B 0,C 180,E1 -19765.892,E2 -19765.892} C_VEL
LIN {X 0,Y 237.927,Z 326.165,A -85,B 0,C 180,E1 -19766.083,E2 -19766.083} C_VEL
LIN {X 0,Y 235.811,Z 323.88,A -85,B 0,C 180,E1 -19766.748,E2 -19766.748} C_VEL
LIN {X 0,Y 234.935,Z 321.224,A -85,B 0,C 180,E1 -19767.136,E2 -19767.136} C_VEL
LIN {X 0,Y 234.889,Z 321.219,A -85,B 0,C 180,E1 -19771.398,E2 -19771.398} C_VEL
LIN {X 0,Y 234.941,Z 321.21,A -85,B 0,C 180,E1 -19775.242,E2 -19775.242} C_VEL
LIN {X 0,Y 234.985,Z 321.202,A -85,B 0,C 180,E1 -19778.968,E2 -19778.968} C_VEL
LIN {X 0,Y 235.084,Z 321.189,A -85,B 0,C 180,E1 -19783.059,E2 -19783.059} C_VEL
LIN {X 0,Y 235.102,Z 321.185,A -85,B 0,C 180,E1 -19787.922,E2 -19787.922} C_VEL
LIN {X 0,Y 235.307,Z 321.169,A -85,B 0,C 180,E1 -19791.412,E2 -19791.412} C_VEL
LIN {X 0,Y 235.344,Z 321.153,A -85,B 0,C 180,E1 -19793.14,E2 -19793.14} C_VEL
LIN {X 0,Y 235.582,Z 321.123,A -85,B 0,C 180,E1 -19798.291,E2 -19798.291} C_VEL
LIN {X 0,Y 235.583,Z 321.133,A -85,B 0,C 180,E1 -19801.71,E2 -19801.71} C_VEL
LIN {X 0,Y 235.392,Z 321.157,A -85,B 0,C 180,E1 -19806.859,E2 -19806.859} C_VEL
LIN {X 0,Y 235.226,Z 321.178,A -85,B 0,C 180,E1 -19810.327,E2 -19810.327} C_VEL
LIN {X 0,Y 235.102,Z 321.196,A -85,B 0,C 180,E1 -19815.608,E2 -19815.608} C_VEL
LIN {X 0,Y 234.997,Z 321.198,A -85,B 0,C 180,E1 -19819.207,E2 -19819.207} C_VEL
LIN {X 0,Y 234.965,Z 321.21,A -85,B 0,C 180,E1 -19822.319,E2 -19822.319} C_VEL
LIN {X 0,Y 234.262,Z 321.293,A -85,B 0,C 180,E1 -19823.75,E2 -19823.75} C_VEL
LIN {X 0,Y 231.412,Z 321.66,A -85,B 0,C 180,E1 -19826.086,E2 -19826.086} C_VEL
LIN {X 0,Y 229.013,Z 321.955,A -85,B 0,C 180,E1 -19827.989,E2 -19827.989} C_VEL
LIN {X 0,Y 227.984,Z 322.082,A -85,B 0,C 180,E1 -19829.466,E2 -19829.466} C_VEL
LIN {X 0,Y 227.899,Z 322.096,A -85,B 0,C 180,E1 -19829.967,E2 -19829.967} C_VEL
LIN {X 0,Y 227.881,Z 322.1,A -85,B 0,C 180,E1 -19833.72,E2 -19833.72} C_VEL
LIN {X 0,Y 227.863,Z 322.103,A -85,B 0,C 180,E1 -19838.088,E2 -19838.088} C_VEL
LIN {X 0,Y 227.883,Z 322.17,A -85,B 0,C 180,E1 -19840.581,E2 -19840.581} C_VEL
LIN {X 0,Y 230.345,Z 329.968,A -85,B 0,C 180,E1 -19845.437,E2 -19845.437} C_VEL
LIN {X 0,Y 231.264,Z 332.771,A -85,B 0,C 180,E1 -19846.941,E2 -19846.941} C_VEL
LIN {X 0,Y 234.141,Z 337.524,A -85,B 0,C 180,E1 -19847.958,E2 -19847.958} C_VEL
LIN {X 0,Y 238.808,Z 345.351,A -85,B 0,C 180,E1 -19849.52,E2 -19849.52} C_VEL
LIN {X 0,Y 243.745,Z 353.993,A -85,B 0,C 180,E1 -19851.07,E2 -19851.07} C_VEL
LIN {X 0,Y 250.222,Z 366.935,A -85,B 0,C 180,E1 -19853.009,E2 -19853.009} C_VEL
LIN {X 0,Y 255.063,Z 377.871,A -85,B 0,C 180,E1 -19854.402,E2 -19854.402} C_VEL
LIN {X 0,Y 257.291,Z 393.04,A -85,B 0,C 180,E1 -19855.385,E2 -19855.385} C_VEL
LIN {X 0,Y 254.759,Z 442.493,A -85,B 0,C 180,E1 -19856.754,E2 -19856.754} C_VEL
LIN {X 0,Y 253.273,Z 456.31,A -85,B 0,C 180,E1 -19857.422,E2 -19857.422} C_VEL
LIN {X 0,Y 251.309,Z 468.209,A -85,B 0,C 180,E1 -19858.261,E2 -19858.261} C_VEL
LIN {X 0,Y 248.625,Z 480.317,A -85,B 0,C 180,E1 -19859.418,E2 -19859.418} C_VEL
LIN {X 0,Y 245.58,Z 491.809,A -85,B 0,C 180,E1 -19860.892,E2 -19860.892} C_VEL
LIN {X 0,Y 242.492,Z 502.171,A -85,B 0,C 180,E1 -19862.61,E2 -19862.61} C_VEL
LIN {X 0,Y 239.671,Z 510.667,A -85,B 0,C 180,E1 -19864.375,E2 -19864.375} C_VEL
LIN {X 0,Y 236.697,Z 518.534,A -85,B 0,C 180,E1 -19866.372,E2 -19866.372} C_VEL
LIN {X 0,Y 233.739,Z 526.252,A -85,B 0,C 180,E1 -19868.853,E2 -19868.853} C_VEL
LIN {X 0,Y 231.425,Z 532.467,A -85,B 0,C 180,E1 -19871.408,E2 -19871.408} C_VEL
LIN {X 0,Y 229.249,Z 537.443,A -85,B 0,C 180,E1 -19873.987,E2 -19873.987} C_VEL
LIN {X 0,Y 227.66,Z 541.317,A -85,B 0,C 180,E1 -19876.616,E2 -19876.616} C_VEL
LIN {X 0,Y 226.607,Z 544.193,A -85,B 0,C 180,E1 -19879.278,E2 -19879.278} C_VEL
LIN {X 0,Y 225.822,Z 546.565,A -85,B 0,C 180,E1 -19882.852,E2 -19882.852} C_VEL
LIN {X 0,Y 225.676,Z 547.278,A -85,B 0,C 180,E1 -19885.242,E2 -19885.242} C_VEL
LIN {X 0,Y 225.721,Z 547.174,A -85,B 0,C 180,E1 -19888.218,E2 -19888.218} C_VEL
LIN {X 0,Y 225.82,Z 546.578,A -85,B 0,C 180,E1 -19890.003,E2 -19890.003} C_VEL
LIN {X 0,Y 225.77,Z 545.579,A -85,B 0,C 180,E1 -19891.786,E2 -19891.786} C_VEL
LIN {X 0,Y 225.723,Z 542.804,A -85,B 0,C 180,E1 -19894.9,E2 -19894.9} C_VEL
LIN {X 0,Y 225.975,Z 538.56,A -85,B 0,C 180,E1 -19898.048,E2 -19898.048} C_VEL
LIN {X 0,Y 226.463,Z 533.719,A -85,B 0,C 180,E1 -19900.734,E2 -19900.734} C_VEL
LIN {X 0,Y 227.285,Z 527.583,A -85,B 0,C 180,E1 -19903.412,E2 -19903.412} C_VEL
LIN {X 0,Y 228.614,Z 519.943,A -85,B 0,C 180,E1 -19906.064,E2 -19906.064} C_VEL
LIN {X 0,Y 230.155,Z 511.498,A -85,B 0,C 180,E1 -19908.404,E2 -19908.404} C_VEL
LIN {X 0,Y 231.97,Z 501.456,A -85,B 0,C 180,E1 -19910.625,E2 -19910.625} C_VEL
LIN {X 0,Y 233.275,Z 493.18,A -85,B 0,C 180,E1 -19912.125,E2 -19912.125} C_VEL
LIN {X 0,Y 234.953,Z 483.229,A -85,B 0,C 180,E1 -19913.586,E2 -19913.586} C_VEL
LIN {X 0,Y 236.715,Z 470.57,A -85,B 0,C 180,E1 -19915.032,E2 -19915.032} C_VEL
LIN {X 0,Y 238.147,Z 457.539,A -85,B 0,C 180,E1 -19916.1,E2 -19916.1} C_VEL
LIN {X 0,Y 239.152,Z 444.717,A -85,B 0,C 180,E1 -19916.804,E2 -19916.804} C_VEL
LIN {X 0,Y 240.511,Z 408.143,A -85,B 0,C 180,E1 -19917.915,E2 -19917.915} C_VEL
LIN {X 0,Y 240.947,Z 386.175,A -85,B 0,C 180,E1 -19918.578,E2 -19918.578} C_VEL
LIN {X 0,Y 236.692,Z 351.248,A -85,B 0,C 180,E1 -19920.166,E2 -19920.166} C_VEL
LIN {X 0,Y 231.445,Z 337.081,A -85,B 0,C 180,E1 -19921.241,E2 -19921.241} C_VEL
LIN {X 0,Y 230.55,Z 334.432,A -85,B 0,C 180,E1 -19921.497,E2 -19921.497} C_VEL
LIN {X 0,Y 228.292,Z 323.834,A -85,B 0,C 180,E1 -19925.8,E2 -19925.8} C_VEL
LIN {X 0,Y 227.916,Z 322.093,A -85,B 0,C 180,E1 -19926.542,E2 -19926.542} C_VEL
LIN {X 0,Y 227.832,Z 322.107,A -85,B 0,C 180,E1 -19930.378,E2 -19930.378} C_VEL
LIN {X 0,Y 227.833,Z 322.105,A -85,B 0,C 180,E1 -19935.196,E2 -19935.196} C_VEL
LIN {X 0,Y 227.832,Z 322.101,A -85,B 0,C 180,E1 -19939.624,E2 -19939.624} C_VEL
LIN {X 0,Y 227.888,Z 322.095,A -85,B 0,C 180,E1 -19944.129,E2 -19944.129} C_VEL
LIN {X 0,Y 227.879,Z 322.096,A -85,B 0,C 180,E1 -19948.379,E2 -19948.379} C_VEL
LIN {X 0,Y 227.895,Z 322.095,A -85,B 0,C 180,E1 -19952.446,E2 -19952.446} C_VEL
LIN {X 0,Y 227.914,Z 322.093,A -85,B 0,C 180,E1 -19956.367,E2 -19956.367} C_VEL
LIN {X 0,Y 227.928,Z 322.081,A -85,B 0,C 180,E1 -19960.173,E2 -19960.173} C_VEL
LIN {X 0,Y 228.029,Z 322.072,A -85,B 0,C 180,E1 -19963.895,E2 -19963.895} C_VEL
LIN {X 0,Y 228.073,Z 322.076,A -85,B 0,C 180,E1 -19967.543,E2 -19967.543} C_VEL
LIN {X 0,Y 228.261,Z 322.042,A -85,B 0,C 180,E1 -19971.144,E2 -19971.144} C_VEL
LIN {X 0,Y 228.31,Z 322.023,A -85,B 0,C 180,E1 -19972.927,E2 -19972.927} C_VEL
LIN {X 0,Y 228.559,Z 322.014,A -85,B 0,C 180,E1 -19978.238,E2 -19978.238} C_VEL
LIN {X 0,Y 228.56,Z 322.011,A -85,B 0,C 180,E1 -19981.762,E2 -19981.762} C_VEL
LIN {X 0,Y 228.325,Z 322.024,A -85,B 0,C 180,E1 -19987.072,E2 -19987.072} C_VEL
LIN {X 0,Y 228.152,Z 322.064,A -85,B 0,C 180,E1 -19990.65,E2 -19990.65} C_VEL
LIN {X 0,Y 228.049,Z 322.077,A -85,B 0,C 180,E1 -19994.273,E2 -19994.273} C_VEL
LIN {X 0,Y 227.959,Z 322.087,A -85,B 0,C 180,E1 -19997.957,E2 -19997.957} C_VEL
LIN {X 0,Y 227.922,Z 322.088,A -85,B 0,C 180,E1 -20002.319,E2 -20002.319} C_VEL
LIN {X 0,Y 227.95,Z 322.09,A -85,B 0,C 180,E1 -20006.601,E2 -20006.601} C_VEL
LIN {X 0,Y 227.915,Z 322.089,A -85,B 0,C 180,E1 -20010.295,E2 -20010.295} C_VEL
LIN {X 0,Y 227.883,Z 322.092,A -85,B 0,C 180,E1 -20013.719,E2 -20013.719} C_VEL
LIN {X 0,Y 227.85,Z 322.098,A -85,B 0,C 180,E1 -20018.089,E2 -20018.089} C_VEL
LIN {X 0,Y 227.817,Z 322.103,A -85,B 0,C 180,E1 -20022.741,E2 -20022.741} C_VEL
LIN {X 0,Y 227.812,Z 322.104,A -85,B 0,C 180,E1 -20027.255,E2 -20027.255} C_VEL
LIN {X 0,Y 227.849,Z 322.103,A -85,B 0,C 180,E1 -20031.907,E2 -20031.907} C_VEL
LIN {X 0,Y 227.884,Z 322.099,A -85,B 0,C 180,E1 -20036.375,E2 -20036.375} C_VEL
LIN {X 0,Y 227.908,Z 322.096,A -85,B 0,C 180,E1 -20040.434,E2 -20040.434} C_VEL
LIN {X 0,Y 227.933,Z 322.092,A -85,B 0,C 180,E1 -20044.424,E2 -20044.424} C_VEL
LIN {X 0,Y 227.995,Z 322.086,A -85,B 0,C 180,E1 -20048.288,E2 -20048.288} C_VEL
LIN {X 0,Y 228.093,Z 322.25,A -85,B 0,C 180,E1 -20053.443,E2 -20053.443} C_VEL
LIN {X 0,Y 229.144,Z 325.022,A -85,B 0,C 180,E1 -20053.668,E2 -20053.668} C_VEL
LIN {X 0,Y 235.419,Z 338.611,A -85,B 0,C 180,E1 -20054.872,E2 -20054.872} C_VEL
LIN {X 0,Y 241.778,Z 356.581,A -85,B 0,C 180,E1 -20056.156,E2 -20056.156} C_VEL
LIN {X 0,Y 240.236,Z 404.641,A -85,B 0,C 180,E1 -20057.55,E2 -20057.55} C_VEL
LIN {X 0,Y 239.352,Z 428.381,A -85,B 0,C 180,E1 -20058.298,E2 -20058.298} C_VEL
LIN {X 0,Y 238.405,Z 441.82,A -85,B 0,C 180,E1 -20059.058,E2 -20059.058} C_VEL
LIN {X 0,Y 237.317,Z 453.937,A -85,B 0,C 180,E1 -20060.086,E2 -20060.086} C_VEL
LIN {X 0,Y 235.771,Z 465.745,A -85,B 0,C 180,E1 -20061.426,E2 -20061.426} C_VEL
LIN {X 0,Y 234.178,Z 477.07,A -85,B 0,C 180,E1 -20063.103,E2 -20063.103} C_VEL
LIN {X 0,Y 232.393,Z 487.324,A -85,B 0,C 180,E1 -20065.01,E2 -20065.01} C_VEL
LIN {X 0,Y 230.588,Z 497.341,A -85,B 0,C 180,E1 -20067.377,E2 -20067.377} C_VEL
LIN {X 0,Y 228.929,Z 506.169,A -85,B 0,C 180,E1 -20069.997,E2 -20069.997} C_VEL
LIN {X 0,Y 227.679,Z 513.2,A -85,B 0,C 180,E1 -20072.651,E2 -20072.651} C_VEL
LIN {X 0,Y 226.835,Z 518.819,A -85,B 0,C 180,E1 -20075.331,E2 -20075.331} C_VEL
LIN {X 0,Y 226.187,Z 523.247,A -85,B 0,C 180,E1 -20078.035,E2 -20078.035} C_VEL
LIN {X 0,Y 225.667,Z 526.599,A -85,B 0,C 180,E1 -20080.767,E2 -20080.767} C_VEL
LIN {X 0,Y 225.514,Z 528.266,A -85,B 0,C 180,E1 -20082.598,E2 -20082.598} C_VEL
LIN {X 0,Y 225.48,Z 529.754,A -85,B 0,C 180,E1 -20084.931,E2 -20084.931} C_VEL
LIN {X 0,Y 225.602,Z 530.693,A -85,B 0,C 180,E1 -20088.148,E2 -20088.148} C_VEL
LIN {X 0,Y 226.19,Z 530.407,A -85,B 0,C 180,E1 -20091.231,E2 -20091.231} C_VEL
LIN {X 0,Y 226.927,Z 529.302,A -85,B 0,C 180,E1 -20093.738,E2 -20093.738} C_VEL
LIN {X 0,Y 228.272,Z 526.883,A -85,B 0,C 180,E1 -20096.768,E2 -20096.768} C_VEL
LIN {X 0,Y 229.759,Z 523.872,A -85,B 0,C 180,E1 -20099.299,E2 -20099.299} C_VEL
LIN {X 0,Y 231.917,Z 519.144,A -85,B 0,C 180,E1 -20102.211,E2 -20102.211} C_VEL
LIN {X 0,Y 234.305,Z 513.719,A -85,B 0,C 180,E1 -20104.74,E2 -20104.74} C_VEL
LIN {X 0,Y 237.188,Z 506.728,A -85,B 0,C 180,E1 -20107.293,E2 -20107.293} C_VEL
LIN {X 0,Y 240.103,Z 498.918,A -85,B 0,C 180,E1 -20109.538,E2 -20109.538} C_VEL
LIN {X 0,Y 243.209,Z 489.688,A -85,B 0,C 180,E1 -20111.65,E2 -20111.65} C_VEL
LIN {X 0,Y 246.355,Z 479.471,A -85,B 0,C 180,E1 -20113.487,E2 -20113.487} C_VEL
LIN {X 0,Y 249.129,Z 468.684,A -85,B 0,C 180,E1 -20115.015,E2 -20115.015} C_VEL
LIN {X 0,Y 251.717,Z 456.02,A -85,B 0,C 180,E1 -20116.394,E2 -20116.394} C_VEL
LIN {X 0,Y 253.683,Z 443.707,A -85,B 0,C 180,E1 -20117.378,E2 -20117.378} C_VEL
LIN {X 0,Y 255.197,Z 430.287,A -85,B 0,C 180,E1 -20118.089,E2 -20118.089} C_VEL
LIN {X 0,Y 256.352,Z 411.59,A -85,B 0,C 180,E1 -20118.653,E2 -20118.653} C_VEL
LIN {X 0,Y 258.135,Z 373.577,A -85,B 0,C 180,E1 -20119.7,E2 -20119.7} C_VEL
LIN {X 0,Y 253.213,Z 363.076,A -85,B 0,C 180,E1 -20121.058,E2 -20121.058} C_VEL
LIN {X 0,Y 246.848,Z 351.124,A -85,B 0,C 180,E1 -20122.879,E2 -20122.879} C_VEL
LIN {X 0,Y 241.543,Z 342.292,A -85,B 0,C 180,E1 -20124.476,E2 -20124.476} C_VEL
LIN {X 0,Y 236.891,Z 335.498,A -85,B 0,C 180,E1 -20125.938,E2 -20125.938} C_VEL
LIN {X 0,Y 234.182,Z 331.63,A -85,B 0,C 180,E1 -20126.836,E2 -20126.836} C_VEL
LIN {X 0,Y 231.826,Z 328.462,A -85,B 0,C 180,E1 -20127.639,E2 -20127.639} C_VEL
LIN {X 0,Y 230.952,Z 327.107,A -85,B 0,C 180,E1 -20127.952,E2 -20127.952} C_VEL
LIN {X 0,Y 228.85,Z 324.957,A -85,B 0,C 180,E1 -20128.671,E2 -20128.671} C_VEL
LIN {X 0,Y 227.943,Z 322.716,A -85,B 0,C 180,E1 -20129.053,E2 -20129.053} C_VEL
LIN {X 0,Y 227.836,Z 322.099,A -85,B 0,C 180,E1 -20129.132,E2 -20129.132} C_VEL
LIN {X 0,Y 227.91,Z 322.097,A -85,B 0,C 180,E1 -20133.407,E2 -20133.407} C_VEL
LIN {X 0,Y 227.943,Z 322.083,A -85,B 0,C 180,E1 -20138.286,E2 -20138.286} C_VEL
LIN {X 0,Y 228.022,Z 322.069,A -85,B 0,C 180,E1 -20142.825,E2 -20142.825} C_VEL
LIN {X 0,Y 228.06,Z 322.063,A -85,B 0,C 180,E1 -20147.543,E2 -20147.543} C_VEL
LIN {X 0,Y 228.246,Z 322.052,A -85,B 0,C 180,E1 -20151.144,E2 -20151.144} C_VEL
LIN {X 0,Y 228.296,Z 322.03,A -85,B 0,C 180,E1 -20152.927,E2 -20152.927} C_VEL
LIN {X 0,Y 228.54,Z 321.999,A -85,B 0,C 180,E1 -20158.238,E2 -20158.238} C_VEL
LIN {X 0,Y 228.542,Z 322.009,A -85,B 0,C 180,E1 -20161.763,E2 -20161.763} C_VEL
LIN {X 0,Y 228.343,Z 322.033,A -85,B 0,C 180,E1 -20167.072,E2 -20167.072} C_VEL
LIN {X 0,Y 228.151,Z 322.062,A -85,B 0,C 180,E1 -20170.651,E2 -20170.651} C_VEL
LIN {X 0,Y 228.053,Z 322.061,A -85,B 0,C 180,E1 -20174.273,E2 -20174.273} C_VEL
LIN {X 0,Y 227.992,Z 322.073,A -85,B 0,C 180,E1 -20177.955,E2 -20177.955} C_VEL
LIN {X 0,Y 227.919,Z 322.087,A -85,B 0,C 180,E1 -20182.331,E2 -20182.331} C_VEL
LIN {X 0,Y 227.933,Z 322.089,A -85,B 0,C 180,E1 -20186.605,E2 -20186.605} C_VEL
LIN {X 0,Y 227.899,Z 322.096,A -85,B 0,C 180,E1 -20189.967,E2 -20189.967} C_VEL
LIN {X 0,Y 227.226,Z 322.188,A -85,B 0,C 180,E1 -20191.442,E2 -20191.442} C_VEL
LIN {X 0,Y 224.37,Z 322.547,A -85,B 0,C 180,E1 -20193.849,E2 -20193.849} C_VEL
LIN {X 0,Y 221.943,Z 322.845,A -85,B 0,C 180,E1 -20195.813,E2 -20195.813} C_VEL
LIN {X 0,Y 220.899,Z 322.972,A -85,B 0,C 180,E1 -20197.337,E2 -20197.337} C_VEL
LIN {X 0,Y 220.813,Z 322.979,A -85,B 0,C 180,E1 -20197.854,E2 -20197.854} C_VEL
LIN {X 0,Y 220.839,Z 323.066,A -85,B 0,C 180,E1 -20198.649,E2 -20198.649} C_VEL
LIN {X 0,Y 222.812,Z 329.387,A -85,B 0,C 180,E1 -20202.949,E2 -20202.949} C_VEL
LIN {X 0,Y 223.742,Z 332.231,A -85,B 0,C 180,E1 -20204.655,E2 -20204.655} C_VEL
LIN {X 0,Y 226.809,Z 337.05,A -85,B 0,C 180,E1 -20205.845,E2 -20205.845} C_VEL
LIN {X 0,Y 228.329,Z 339.402,A -85,B 0,C 180,E1 -20206.411,E2 -20206.411} C_VEL
LIN {X 0,Y 232.048,Z 345.431,A -85,B 0,C 180,E1 -20207.751,E2 -20207.751} C_VEL
LIN {X 0,Y 237.338,Z 354.567,A -85,B 0,C 180,E1 -20209.551,E2 -20209.551} C_VEL
LIN {X 0,Y 243.562,Z 366.562,A -85,B 0,C 180,E1 -20211.543,E2 -20211.543} C_VEL
LIN {X 0,Y 249.869,Z 380.613,A -85,B 0,C 180,E1 -20213.464,E2 -20213.464} C_VEL
LIN {X 0,Y 251.834,Z 394.305,A -85,B 0,C 180,E1 -20214.382,E2 -20214.382} C_VEL
LIN {X 0,Y 249.255,Z 442.441,A -85,B 0,C 180,E1 -20215.737,E2 -20215.737} C_VEL
LIN {X 0,Y 247.697,Z 456.189,A -85,B 0,C 180,E1 -20216.411,E2 -20216.411} C_VEL
LIN {X 0,Y 245.561,Z 468.598,A -85,B 0,C 180,E1 -20217.306,E2 -20217.306} C_VEL
LIN {X 0,Y 242.981,Z 479.721,A -85,B 0,C 180,E1 -20218.386,E2 -20218.386} C_VEL
LIN {X 0,Y 239.825,Z 491.264,A -85,B 0,C 180,E1 -20219.881,E2 -20219.881} C_VEL
LIN {X 0,Y 236.641,Z 501.663,A -85,B 0,C 180,E1 -20221.632,E2 -20221.632} C_VEL
LIN {X 0,Y 233.324,Z 511.075,A -85,B 0,C 180,E1 -20223.625,E2 -20223.625} C_VEL
LIN {X 0,Y 229.64,Z 520.175,A -85,B 0,C 180,E1 -20226.08,E2 -20226.08} C_VEL
LIN {X 0,Y 226.742,Z 527.448,A -85,B 0,C 180,E1 -20228.612,E2 -20228.612} C_VEL
LIN {X 0,Y 223.899,Z 534.333,A -85,B 0,C 180,E1 -20231.709,E2 -20231.709} C_VEL
LIN {X 0,Y 221.784,Z 538.855,A -85,B 0,C 180,E1 -20234.377,E2 -20234.377} C_VEL
LIN {X 0,Y 220.305,Z 542.32,A -85,B 0,C 180,E1 -20237.1,E2 -20237.1} C_VEL
LIN {X 0,Y 219.093,Z 545.412,A -85,B 0,C 180,E1 -20240.773,E2 -20240.773} C_VEL
LIN {X 0,Y 218.573,Z 546.95,A -85,B 0,C 180,E1 -20244.467,E2 -20244.467} C_VEL
LIN {X 0,Y 218.558,Z 547.102,A -85,B 0,C 180,E1 -20246.315,E2 -20246.315} C_VEL
LIN {X 0,Y 218.633,Z 546.864,A -85,B 0,C 180,E1 -20248.161,E2 -20248.161} C_VEL
LIN {X 0,Y 218.752,Z 546.239,A -85,B 0,C 180,E1 -20250.003,E2 -20250.003} C_VEL
LIN {X 0,Y 218.681,Z 545.208,A -85,B 0,C 180,E1 -20251.844,E2 -20251.844} C_VEL
LIN {X 0,Y 218.624,Z 542.673,A -85,B 0,C 180,E1 -20254.76,E2 -20254.76} C_VEL
LIN {X 0,Y 218.832,Z 539.417,A -85,B 0,C 180,E1 -20257.384,E2 -20257.384} C_VEL
LIN {X 0,Y 219.239,Z 534.902,A -85,B 0,C 180,E1 -20260.158,E2 -20260.158} C_VEL
LIN {X 0,Y 220.148,Z 528.024,A -85,B 0,C 180,E1 -20263.385,E2 -20263.385} C_VEL
LIN {X 0,Y 221.52,Z 520.537,A -85,B 0,C 180,E1 -20266.12,E2 -20266.12} C_VEL
LIN {X 0,Y 223.182,Z 511.568,A -85,B 0,C 180,E1 -20268.731,E2 -20268.731} C_VEL
LIN {X 0,Y 225.087,Z 501.449,A -85,B 0,C 180,E1 -20271.046,E2 -20271.046} C_VEL
LIN {X 0,Y 226.729,Z 491.927,A -85,B 0,C 180,E1 -20272.8,E2 -20272.8} C_VEL
LIN {X 0,Y 228.386,Z 481.73,A -85,B 0,C 180,E1 -20274.307,E2 -20274.307} C_VEL
LIN {X 0,Y 230.099,Z 469.749,A -85,B 0,C 180,E1 -20275.682,E2 -20275.682} C_VEL
LIN {X 0,Y 231.531,Z 457.218,A -85,B 0,C 180,E1 -20276.722,E2 -20276.722} C_VEL
LIN {X 0,Y 232.557,Z 443.929,A -85,B 0,C 180,E1 -20277.468,E2 -20277.468} C_VEL
LIN {X 0,Y 234.239,Z 396.996,A -85,B 0,C 180,E1 -20278.912,E2 -20278.912} C_VEL
LIN {X 0,Y 234.395,Z 386.88,A -85,B 0,C 180,E1 -20279.232,E2 -20279.232} C_VEL
LIN {X 0,Y 230.37,Z 353.145,A -85,B 0,C 180,E1 -20280.818,E2 -20280.818} C_VEL
LIN {X 0,Y 224.467,Z 337.416,A -85,B 0,C 180,E1 -20282.082,E2 -20282.082} C_VEL
LIN {X 0,Y 223.322,Z 334.293,A -85,B 0,C 180,E1 -20282.346,E2 -20282.346} C_VEL
LIN {X 0,Y 221.157,Z 324.282,A -85,B 0,C 180,E1 -20286.576,E2 -20286.576} C_VEL
LIN {X 0,Y 220.832,Z 322.978,A -85,B 0,C 180,E1 -20287.209,E2 -20287.209} C_VEL
LIN {X 0,Y 220.774,Z 322.984,A -85,B 0,C 180,E1 -20291.955,E2 -20291.955} C_VEL
LIN {X 0,Y 220.775,Z 322.983,A -85,B 0,C 180,E1 -20295.546,E2 -20295.546} C_VEL
LIN {X 0,Y 220.814,Z 322.977,A -85,B 0,C 180,E1 -20300.464,E2 -20300.464} C_VEL
LIN {X 0,Y 220.809,Z 322.977,A -85,B 0,C 180,E1 -20305.046,E2 -20305.046} C_VEL
LIN {X 0,Y 220.877,Z 322.966,A -85,B 0,C 180,E1 -20309.396,E2 -20309.396} C_VEL
LIN {X 0,Y 220.903,Z 322.969,A -85,B 0,C 180,E1 -20313.55,E2 -20313.55} C_VEL
LIN {X 0,Y 220.872,Z 322.971,A -85,B 0,C 180,E1 -20317.552,E2 -20317.552} C_VEL
LIN {X 0,Y 220.932,Z 322.947,A -85,B 0,C 180,E1 -20322.622,E2 -20322.622} C_VEL
LIN {X 0,Y 221.01,Z 322.953,A -85,B 0,C 180,E1 -20327.138,E2 -20327.138} C_VEL
LIN {X 0,Y 221.202,Z 322.92,A -85,B 0,C 180,E1 -20330.859,E2 -20330.859} C_VEL
LIN {X 0,Y 221.131,Z 322.921,A -85,B 0,C 180,E1 -20334.528,E2 -20334.528} C_VEL
LIN {X 0,Y 221.517,Z 322.891,A -85,B 0,C 180,E1 -20338.181,E2 -20338.181} C_VEL
LIN {X 0,Y 221.518,Z 322.887,A -85,B 0,C 180,E1 -20341.818,E2 -20341.818} C_VEL
LIN {X 0,Y 221.261,Z 322.904,A -85,B 0,C 180,E1 -20347.299,E2 -20347.299} C_VEL
LIN {X 0,Y 221.073,Z 322.945,A -85,B 0,C 180,E1 -20350.996,E2 -20350.996} C_VEL
LIN {X 0,Y 220.976,Z 322.954,A -85,B 0,C 180,E1 -20354.74,E2 -20354.74} C_VEL
LIN {X 0,Y 220.895,Z 322.969,A -85,B 0,C 180,E1 -20358.551,E2 -20358.551} C_VEL
LIN {X 0,Y 220.891,Z 322.964,A -85,B 0,C 180,E1 -20362.673,E2 -20362.673} C_VEL
LIN {X 0,Y 220.892,Z 322.967,A -85,B 0,C 180,E1 -20367.014,E2 -20367.014} C_VEL
LIN {X 0,Y 220.87,Z 322.968,A -85,B 0,C 180,E1 -20370.777,E2 -20370.777} C_VEL
LIN {X 0,Y 220.807,Z 322.973,A -85,B 0,C 180,E1 -20374.953,E2 -20374.953} C_VEL
LIN {X 0,Y 220.813,Z 322.973,A -85,B 0,C 180,E1 -20379.535,E2 -20379.535} C_VEL
LIN {X 0,Y 220.777,Z 322.978,A -85,B 0,C 180,E1 -20384.453,E2 -20384.453} C_VEL
LIN {X 0,Y 220.772,Z 322.983,A -85,B 0,C 180,E1 -20388.045,E2 -20388.045} C_VEL
LIN {X 0,Y 220.811,Z 322.975,A -85,B 0,C 180,E1 -20390.461,E2 -20390.461} C_VEL
LIN {X 0,Y 220.806,Z 322.976,A -85,B 0,C 180,E1 -20395.043,E2 -20395.043} C_VEL
LIN {X 0,Y 220.838,Z 322.974,A -85,B 0,C 180,E1 -20399.388,E2 -20399.388} C_VEL
LIN {X 0,Y 220.898,Z 322.968,A -85,B 0,C 180,E1 -20403.547,E2 -20403.547} C_VEL
LIN {X 0,Y 220.928,Z 322.965,A -85,B 0,C 180,E1 -20407.556,E2 -20407.556} C_VEL
LIN {X 0,Y 221.002,Z 322.971,A -85,B 0,C 180,E1 -20412.557,E2 -20412.557} C_VEL
LIN {X 0,Y 222.019,Z 325.844,A -85,B 0,C 180,E1 -20412.795,E2 -20412.795} C_VEL
LIN {X 0,Y 229.03,Z 340.525,A -85,B 0,C 180,E1 -20414.19,E2 -20414.19} C_VEL
LIN {X 0,Y 235.303,Z 358.098,A -85,B 0,C 180,E1 -20415.511,E2 -20415.511} C_VEL
LIN {X 0,Y 232.808,Z 427.939,A -85,B 0,C 180,E1 -20417.631,E2 -20417.631} C_VEL
LIN {X 0,Y 231.817,Z 441.624,A -85,B 0,C 180,E1 -20418.411,E2 -20418.411} C_VEL
LIN {X 0,Y 230.682,Z 453.892,A -85,B 0,C 180,E1 -20419.465,E2 -20419.465} C_VEL
LIN {X 0,Y 228.967,Z 466.559,A -85,B 0,C 180,E1 -20420.947,E2 -20420.947} C_VEL
LIN {X 0,Y 227.319,Z 477.783,A -85,B 0,C 180,E1 -20422.67,E2 -20422.67} C_VEL
LIN {X 0,Y 225.473,Z 487.93,A -85,B 0,C 180,E1 -20424.632,E2 -20424.632} C_VEL
LIN {X 0,Y 223.782,Z 497.067,A -85,B 0,C 180,E1 -20426.847,E2 -20426.847} C_VEL
LIN {X 0,Y 222.018,Z 505.991,A -85,B 0,C 180,E1 -20429.544,E2 -20429.544} C_VEL
LIN {X 0,Y 220.712,Z 513.131,A -85,B 0,C 180,E1 -20432.278,E2 -20432.278} C_VEL
LIN {X 0,Y 219.675,Z 519.637,A -85,B 0,C 180,E1 -20435.505,E2 -20435.505} C_VEL
LIN {X 0,Y 219.035,Z 523.941,A -85,B 0,C 180,E1 -20438.299,E2 -20438.299} C_VEL
LIN {X 0,Y 218.519,Z 527.177,A -85,B 0,C 180,E1 -20441.123,E2 -20441.123} C_VEL
LIN {X 0,Y 218.421,Z 528.786,A -85,B 0,C 180,E1 -20443.014,E2 -20443.014} C_VEL
LIN {X 0,Y 218.388,Z 530.023,A -85,B 0,C 180,E1 -20445.109,E2 -20445.109} C_VEL
LIN {X 0,Y 218.579,Z 530.995,A -85,B 0,C 180,E1 -20448.752,E2 -20448.752} C_VEL
LIN {X 0,Y 219.168,Z 530.684,A -85,B 0,C 180,E1 -20451.576,E2 -20451.576} C_VEL
LIN {X 0,Y 220.107,Z 529.377,A -85,B 0,C 180,E1 -20454.522,E2 -20454.522} C_VEL
LIN {X 0,Y 221.406,Z 527.188,A -85,B 0,C 180,E1 -20457.279,E2 -20457.279} C_VEL
LIN {X 0,Y 223.218,Z 523.704,A -85,B 0,C 180,E1 -20460.245,E2 -20460.245} C_VEL
LIN {X 0,Y 225.437,Z 519.188,A -85,B 0,C 180,E1 -20463.035,E2 -20463.035} C_VEL
LIN {X 0,Y 228.187,Z 513.266,A -85,B 0,C 180,E1 -20465.812,E2 -20465.812} C_VEL
LIN {X 0,Y 231.371,Z 505.761,A -85,B 0,C 180,E1 -20468.509,E2 -20468.509} C_VEL
LIN {X 0,Y 234.377,Z 498.042,A -85,B 0,C 180,E1 -20470.703,E2 -20470.703} C_VEL
LIN {X 0,Y 237.708,Z 488.6,A -85,B 0,C 180,E1 -20472.84,E2 -20472.84} C_VEL
LIN {X 0,Y 240.978,Z 478.005,A -85,B 0,C 180,E1 -20474.712,E2 -20474.712} C_VEL
LIN {X 0,Y 244.023,Z 466.253,A -85,B 0,C 180,E1 -20476.319,E2 -20476.319} C_VEL
LIN {X 0,Y 246.414,Z 454.548,A -85,B 0,C 180,E1 -20477.555,E2 -20477.555} C_VEL
LIN {X 0,Y 248.506,Z 441.421,A -85,B 0,C 180,E1 -20478.538,E2 -20478.538} C_VEL
LIN {X 0,Y 249.863,Z 428.76,A -85,B 0,C 180,E1 -20479.179,E2 -20479.179} C_VEL
LIN {X 0,Y 252.676,Z 375.902,A -85,B 0,C 180,E1 -20480.681,E2 -20480.681} C_VEL
LIN {X 0,Y 246.429,Z 362.773,A -85,B 0,C 180,E1 -20482.504,E2 -20482.504} C_VEL
LIN {X 0,Y 238.561,Z 348.631,A -85,B 0,C 180,E1 -20484.938,E2 -20484.938} C_VEL
LIN {X 0,Y 232.784,Z 340.202,A -85,B 0,C 180,E1 -20486.824,E2 -20486.824} C_VEL
LIN {X 0,Y 230.483,Z 336.92,A -85,B 0,C 180,E1 -20487.621,E2 -20487.621} C_VEL
LIN {X 0,Y 227.332,Z 332.651,A -85,B 0,C 180,E1 -20488.749,E2 -20488.749} C_VEL
LIN {X 0,Y 224.927,Z 329.528,A -85,B 0,C 180,E1 -20489.644,E2 -20489.644} C_VEL
LIN {X 0,Y 224.289,Z 328.236,A -85,B 0,C 180,E1 -20489.911,E2 -20489.911} C_VEL
LIN {X 0,Y 221.915,Z 326.013,A -85,B 0,C 180,E1 -20490.797,E2 -20490.797} C_VEL
LIN {X 0,Y 220.853,Z 323.421,A -85,B 0,C 180,E1 -20491.294,E2 -20491.294} C_VEL
LIN {X 0,Y 220.78,Z 322.976,A -85,B 0,C 180,E1 -20491.349,E2 -20491.349} C_VEL
LIN {X 0,Y 220.863,Z 322.975,A -85,B 0,C 180,E1 -20493.546,E2 -20493.546} C_VEL
LIN {X 0,Y 220.856,Z 322.973,A -85,B 0,C 180,E1 -20497.551,E2 -20497.551} C_VEL
LIN {X 0,Y 220.972,Z 322.949,A -85,B 0,C 180,E1 -20502.571,E2 -20502.571} C_VEL
LIN {X 0,Y 220.999,Z 322.945,A -85,B 0,C 180,E1 -20507.138,E2 -20507.138} C_VEL
LIN {X 0,Y 221.185,Z 322.933,A -85,B 0,C 180,E1 -20510.859,E2 -20510.859} C_VEL
LIN {X 0,Y 221.115,Z 322.933,A -85,B 0,C 180,E1 -20514.529,E2 -20514.529} C_VEL
LIN {X 0,Y 221.498,Z 322.876,A -85,B 0,C 180,E1 -20518.182,E2 -20518.182} C_VEL
LIN {X 0,Y 221.499,Z 322.885,A -85,B 0,C 180,E1 -20521.819,E2 -20521.819} C_VEL
LIN {X 0,Y 221.278,Z 322.91,A -85,B 0,C 180,E1 -20527.299,E2 -20527.299} C_VEL
LIN {X 0,Y 221.1,Z 322.943,A -85,B 0,C 180,E1 -20530.995,E2 -20530.995} C_VEL
LIN {X 0,Y 221.005,Z 322.955,A -85,B 0,C 180,E1 -20536.631,E2 -20536.631} C_VEL
LIN {X 0,Y 220.882,Z 322.967,A -85,B 0,C 180,E1 -20540.488,E2 -20540.488} C_VEL
LIN {X 0,Y 220.857,Z 322.962,A -85,B 0,C 180,E1 -20544.437,E2 -20544.437} C_VEL
LIN {X 0,Y 220.827,Z 322.966,A -85,B 0,C 180,E1 -20548.515,E2 -20548.515} C_VEL
LIN {X 0,Y 220.816,Z 322.971,A -85,B 0,C 180,E1 -20552.757,E2 -20552.757} C_VEL
LIN {X 0,Y 220.83,Z 322.98,A -85,B 0,C 180,E1 -20557.29,E2 -20557.29} C_VEL
LIN {X 0,Y 220.813,Z 322.979,A -85,B 0,C 180,E1 -20557.854,E2 -20557.854} C_VEL
LIN {X 0,Y 220.39,Z 323.692,A -85,B 0,C 180,E1 -20558.734,E2 -20558.734} C_VEL
LIN {X 0,Y 218.981,Z 326.145,A -85,B 0,C 180,E1 -20559.831,E2 -20559.831} C_VEL
LIN {X 0,Y 216.758,Z 330.94,A -85,B 0,C 180,E1 -20561.683,E2 -20561.683} C_VEL
LIN {X 0,Y 217.139,Z 333.3,A -85,B 0,C 180,E1 -20562.468,E2 -20562.468} C_VEL
LIN {X 0,Y 217.357,Z 333.712,A -85,B 0,C 180,E1 -20562.582,E2 -20562.582} C_VEL
LIN {X 0,Y 220.786,Z 338.475,A -85,B 0,C 180,E1 -20564.019,E2 -20564.019} C_VEL
LIN {X 0,Y 224.831,Z 344.771,A -85,B 0,C 180,E1 -20565.627,E2 -20565.627} C_VEL
LIN {X 0,Y 228.815,Z 351.39,A -85,B 0,C 180,E1 -20567.125,E2 -20567.125} C_VEL
LIN {X 0,Y 235.147,Z 362.664,A -85,B 0,C 180,E1 -20569.35,E2 -20569.35} C_VEL
LIN {X 0,Y 241.534,Z 376.04,A -85,B 0,C 180,E1 -20571.467,E2 -20571.467} C_VEL
LIN {X 0,Y 244.929,Z 384.065,A -85,B 0,C 180,E1 -20572.554,E2 -20572.554} C_VEL
LIN {X 0,Y 246.466,Z 395.215,A -85,B 0,C 180,E1 -20573.322,E2 -20573.322} C_VEL
LIN {X 0,Y 243.772,Z 442.926,A -85,B 0,C 180,E1 -20574.695,E2 -20574.695} C_VEL
LIN {X 0,Y 242.112,Z 456.815,A -85,B 0,C 180,E1 -20575.403,E2 -20575.403} C_VEL
LIN {X 0,Y 239.885,Z 468.961,A -85,B 0,C 180,E1 -20576.305,E2 -20576.305} C_VEL
LIN {X 0,Y 237.013,Z 480.706,A -85,B 0,C 180,E1 -20577.493,E2 -20577.493} C_VEL
LIN {X 0,Y 233.754,Z 492.022,A -85,B 0,C 180,E1 -20579.014,E2 -20579.014} C_VEL
LIN {X 0,Y 230.444,Z 502.246,A -85,B 0,C 180,E1 -20580.797,E2 -20580.797} C_VEL
LIN {X 0,Y 227.014,Z 511.466,A -85,B 0,C 180,E1 -20582.833,E2 -20582.833} C_VEL
LIN {X 0,Y 223.185,Z 520.445,A -85,B 0,C 180,E1 -20585.343,E2 -20585.343} C_VEL
LIN {X 0,Y 219.964,Z 528.041,A -85,B 0,C 180,E1 -20588.105,E2 -20588.105} C_VEL
LIN {X 0,Y 217.141,Z 534.378,A -85,B 0,C 180,E1 -20591.119,E2 -20591.119} C_VEL
LIN {X 0,Y 214.946,Z 538.826,A -85,B 0,C 180,E1 -20593.867,E2 -20593.867} C_VEL
LIN {X 0,Y 213.345,Z 542.228,A -85,B 0,C 180,E1 -20596.671,E2 -20596.671} C_VEL
LIN {X 0,Y 212.067,Z 545.254,A -85,B 0,C 180,E1 -20600.465,E2 -20600.465} C_VEL
LIN {X 0,Y 211.688,Z 546.185,A -85,B 0,C 180,E1 -20602.372,E2 -20602.372} C_VEL
LIN {X 0,Y 211.473,Z 546.843,A -85,B 0,C 180,E1 -20605.571,E2 -20605.571} C_VEL
LIN {X 0,Y 211.548,Z 546.553,A -85,B 0,C 180,E1 -20608.099,E2 -20608.099} C_VEL
LIN {X 0,Y 211.685,Z 545.899,A -85,B 0,C 180,E1 -20610.003,E2 -20610.003} C_VEL
LIN {X 0,Y 211.595,Z 544.82,A -85,B 0,C 180,E1 -20611.906,E2 -20611.906} C_VEL
LIN {X 0,Y 211.537,Z 542.494,A -85,B 0,C 180,E1 -20614.648,E2 -20614.648} C_VEL
LIN {X 0,Y 211.747,Z 538.909,A -85,B 0,C 180,E1 -20617.632,E2 -20617.632} C_VEL
LIN {X 0,Y 212.195,Z 534.318,A -85,B 0,C 180,E1 -20620.499,E2 -20620.499} C_VEL
LIN {X 0,Y 213.206,Z 527.327,A -85,B 0,C 180,E1 -20623.829,E2 -20623.829} C_VEL
LIN {X 0,Y 214.631,Z 519.742,A -85,B 0,C 180,E1 -20626.652,E2 -20626.652} C_VEL
LIN {X 0,Y 216.162,Z 511.986,A -85,B 0,C 180,E1 -20628.976,E2 -20628.976} C_VEL
LIN {X 0,Y 218.018,Z 502.521,A -85,B 0,C 180,E1 -20631.266,E2 -20631.266} C_VEL
LIN {X 0,Y 219.622,Z 493.262,A -85,B 0,C 180,E1 -20633.082,E2 -20633.082} C_VEL
LIN {X 0,Y 221.401,Z 483.443,A -85,B 0,C 180,E1 -20634.625,E2 -20634.625} C_VEL
LIN {X 0,Y 223.256,Z 470.968,A -85,B 0,C 180,E1 -20636.152,E2 -20636.152} C_VEL
LIN {X 0,Y 224.742,Z 459.142,A -85,B 0,C 180,E1 -20637.219,E2 -20637.219} C_VEL
LIN {X 0,Y 225.883,Z 445.986,A -85,B 0,C 180,E1 -20638.029,E2 -20638.029} C_VEL
LIN {X 0,Y 226.718,Z 427.153,A -85,B 0,C 180,E1 -20638.691,E2 -20638.691} C_VEL
LIN {X 0,Y 227.917,Z 387.797,A -85,B 0,C 180,E1 -20639.91,E2 -20639.91} C_VEL
LIN {X 0,Y 224.093,Z 355.26,A -85,B 0,C 180,E1 -20641.497,E2 -20641.497} C_VEL
LIN {X 0,Y 218.618,Z 340.61,A -85,B 0,C 180,E1 -20642.72,E2 -20642.72} C_VEL
LIN {X 0,Y 215.994,Z 333.855,A -85,B 0,C 180,E1 -20643.384,E2 -20643.384} C_VEL
LIN {X 0,Y 213.947,Z 324.804,A -85,B 0,C 180,E1 -20647.385,E2 -20647.385} C_VEL
LIN {X 0,Y 213.738,Z 323.861,A -85,B 0,C 180,E1 -20647.893,E2 -20647.893} C_VEL
LIN {X 0,Y 213.718,Z 323.864,A -85,B 0,C 180,E1 -20651.127,E2 -20651.127} C_VEL
LIN {X 0,Y 213.71,Z 323.864,A -85,B 0,C 180,E1 -20653.681,E2 -20653.681} C_VEL
LIN {X 0,Y 213.71,Z 323.863,A -85,B 0,C 180,E1 -20656.346,E2 -20656.346} C_VEL
LIN {X 0,Y 213.724,Z 323.859,A -85,B 0,C 180,E1 -20659.144,E2 -20659.144} C_VEL
LIN {X 0,Y 213.752,Z 323.855,A -85,B 0,C 180,E1 -20663.713,E2 -20663.713} C_VEL
LIN {X 0,Y 213.804,Z 323.851,A -85,B 0,C 180,E1 -20668.726,E2 -20668.726} C_VEL
LIN {X 0,Y 213.835,Z 323.847,A -85,B 0,C 180,E1 -20672.604,E2 -20672.604} C_VEL
LIN {X 0,Y 213.827,Z 323.85,A -85,B 0,C 180,E1 -20676.975,E2 -20676.975} C_VEL
LIN {X 0,Y 213.896,Z 323.823,A -85,B 0,C 180,E1 -20682.799,E2 -20682.799} C_VEL
LIN {X 0,Y 213.949,Z 323.832,A -85,B 0,C 180,E1 -20686.706,E2 -20686.706} C_VEL
LIN {X 0,Y 214.142,Z 323.8,A -85,B 0,C 180,E1 -20690.555,E2 -20690.555} C_VEL
LIN {X 0,Y 214.093,Z 323.795,A -85,B 0,C 180,E1 -20694.348,E2 -20694.348} C_VEL
LIN {X 0,Y 214.45,Z 323.77,A -85,B 0,C 180,E1 -20698.122,E2 -20698.122} C_VEL
LIN {X 0,Y 214.554,Z 323.759,A -85,B 0,C 180,E1 -20700,E2 -20700} C_VEL
LIN {X 0,Y 214.451,Z 323.766,A -85,B 0,C 180,E1 -20701.878,E2 -20701.878} C_VEL
LIN {X 0,Y 214.201,Z 323.783,A -85,B 0,C 180,E1 -20707.541,E2 -20707.541} C_VEL
LIN {X 0,Y 214.004,Z 323.825,A -85,B 0,C 180,E1 -20711.364,E2 -20711.364} C_VEL
LIN {X 0,Y 213.91,Z 323.831,A -85,B 0,C 180,E1 -20715.238,E2 -20715.238} C_VEL
LIN {X 0,Y 213.82,Z 323.85,A -85,B 0,C 180,E1 -20719.189,E2 -20719.189} C_VEL
LIN {X 0,Y 213.818,Z 323.847,A -85,B 0,C 180,E1 -20723.23,E2 -20723.23} C_VEL
LIN {X 0,Y 213.836,Z 323.843,A -85,B 0,C 180,E1 -20727.448,E2 -20727.448} C_VEL
LIN {X 0,Y 213.784,Z 323.852,A -85,B 0,C 180,E1 -20731.734,E2 -20731.734} C_VEL
LIN {X 0,Y 213.75,Z 323.853,A -85,B 0,C 180,E1 -20736.287,E2 -20736.287} C_VEL
LIN {X 0,Y 213.718,Z 323.855,A -85,B 0,C 180,E1 -20741.123,E2 -20741.123} C_VEL
LIN {X 0,Y 213.711,Z 323.862,A -85,B 0,C 180,E1 -20743.677,E2 -20743.677} C_VEL
LIN {X 0,Y 213.708,Z 323.86,A -85,B 0,C 180,E1 -20746.343,E2 -20746.343} C_VEL
LIN {X 0,Y 213.721,Z 323.86,A -85,B 0,C 180,E1 -20749.141,E2 -20749.141} C_VEL
LIN {X 0,Y 213.749,Z 323.858,A -85,B 0,C 180,E1 -20753.71,E2 -20753.71} C_VEL
LIN {X 0,Y 213.772,Z 323.854,A -85,B 0,C 180,E1 -20758.26,E2 -20758.26} C_VEL
LIN {X 0,Y 213.83,Z 323.849,A -85,B 0,C 180,E1 -20762.601,E2 -20762.601} C_VEL
LIN {X 0,Y 213.866,Z 323.844,A -85,B 0,C 180,E1 -20766.944,E2 -20766.944} C_VEL
LIN {X 0,Y 213.903,Z 323.841,A -85,B 0,C 180,E1 -20771.601,E2 -20771.601} C_VEL
LIN {X 0,Y 214.984,Z 326.792,A -85,B 0,C 180,E1 -20771.875,E2 -20771.875} C_VEL
LIN {X 0,Y 221.703,Z 340.34,A -85,B 0,C 180,E1 -20773.276,E2 -20773.276} C_VEL
LIN {X 0,Y 226.879,Z 353.83,A -85,B 0,C 180,E1 -20774.394,E2 -20774.394} C_VEL
LIN {X 0,Y 228.896,Z 359.979,A -85,B 0,C 180,E1 -20774.847,E2 -20774.847} C_VEL
LIN {X 0,Y 226.261,Z 427.58,A -85,B 0,C 180,E1 -20776.927,E2 -20776.927} C_VEL
LIN {X 0,Y 225.258,Z 441.428,A -85,B 0,C 180,E1 -20777.726,E2 -20777.726} C_VEL
LIN {X 0,Y 224.096,Z 453.826,A -85,B 0,C 180,E1 -20778.808,E2 -20778.808} C_VEL
LIN {X 0,Y 222.41,Z 465.789,A -85,B 0,C 180,E1 -20780.218,E2 -20780.218} C_VEL
LIN {X 0,Y 220.706,Z 477.195,A -85,B 0,C 180,E1 -20781.989,E2 -20781.989} C_VEL
LIN {X 0,Y 218.708,Z 487.882,A -85,B 0,C 180,E1 -20784.081,E2 -20784.081} C_VEL
LIN {X 0,Y 216.971,Z 496.797,A -85,B 0,C 180,E1 -20786.283,E2 -20786.283} C_VEL
LIN {X 0,Y 215.141,Z 505.806,A -85,B 0,C 180,E1 -20789.061,E2 -20789.061} C_VEL
LIN {X 0,Y 213.75,Z 513.051,A -85,B 0,C 180,E1 -20791.881,E2 -20791.881} C_VEL
LIN {X 0,Y 212.764,Z 518.817,A -85,B 0,C 180,E1 -20794.734,E2 -20794.734} C_VEL
LIN {X 0,Y 212.082,Z 523.362,A -85,B 0,C 180,E1 -20797.614,E2 -20797.614} C_VEL
LIN {X 0,Y 211.678,Z 525.776,A -85,B 0,C 180,E1 -20799.553,E2 -20799.553} C_VEL
LIN {X 0,Y 211.382,Z 527.756,A -85,B 0,C 180,E1 -20801.504,E2 -20801.504} C_VEL
LIN {X 0,Y 211.293,Z 529.276,A -85,B 0,C 180,E1 -20803.461,E2 -20803.461} C_VEL
LIN {X 0,Y 211.28,Z 530.349,A -85,B 0,C 180,E1 -20805.43,E2 -20805.43} C_VEL
LIN {X 0,Y 211.358,Z 531.023,A -85,B 0,C 180,E1 -20807.41,E2 -20807.41} C_VEL
LIN {X 0,Y 211.586,Z 531.291,A -85,B 0,C 180,E1 -20809.397,E2 -20809.397} C_VEL
LIN {X 0,Y 212.169,Z 530.958,A -85,B 0,C 180,E1 -20811.954,E2 -20811.954} C_VEL
LIN {X 0,Y 213.325,Z 529.454,A -85,B 0,C 180,E1 -20815.355,E2 -20815.355} C_VEL
LIN {X 0,Y 214.549,Z 527.499,A -85,B 0,C 180,E1 -20817.818,E2 -20817.818} C_VEL
LIN {X 0,Y 216.765,Z 523.541,A -85,B 0,C 180,E1 -20821.245,E2 -20821.245} C_VEL
LIN {X 0,Y 219.211,Z 518.844,A -85,B 0,C 180,E1 -20824.125,E2 -20824.125} C_VEL
LIN {X 0,Y 222.135,Z 512.766,A -85,B 0,C 180,E1 -20826.947,E2 -20826.947} C_VEL
LIN {X 0,Y 225.6,Z 505.098,A -85,B 0,C 180,E1 -20829.685,E2 -20829.685} C_VEL
LIN {X 0,Y 228.742,Z 497.183,A -85,B 0,C 180,E1 -20831.929,E2 -20831.929} C_VEL
LIN {X 0,Y 232.293,Z 487.452,A -85,B 0,C 180,E1 -20834.092,E2 -20834.092} C_VEL
LIN {X 0,Y 235.705,Z 476.609,A -85,B 0,C 180,E1 -20835.968,E2 -20835.968} C_VEL
LIN {X 0,Y 238.56,Z 465.822,A -85,B 0,C 180,E1 -20837.43,E2 -20837.43} C_VEL
LIN {X 0,Y 241.016,Z 454.084,A -85,B 0,C 180,E1 -20838.661,E2 -20838.661} C_VEL
LIN {X 0,Y 243.058,Z 441.629,A -85,B 0,C 180,E1 -20839.596,E2 -20839.596} C_VEL
LIN {X 0,Y 244.522,Z 428.38,A -85,B 0,C 180,E1 -20840.267,E2 -20840.267} C_VEL
LIN {X 0,Y 247.296,Z 378.325,A -85,B 0,C 180,E1 -20841.7,E2 -20841.7} C_VEL
LIN {X 0,Y 240.96,Z 365.036,A -85,B 0,C 180,E1 -20843.661,E2 -20843.661} C_VEL
LIN {X 0,Y 233.964,Z 352.609,A -85,B 0,C 180,E1 -20845.941,E2 -20845.941} C_VEL
LIN {X 0,Y 227.383,Z 342.823,A -85,B 0,C 180,E1 -20848.237,E2 -20848.237} C_VEL
LIN {X 0,Y 223.654,Z 337.896,A -85,B 0,C 180,E1 -20849.621,E2 -20849.621} C_VEL
LIN {X 0,Y 220.637,Z 333.768,A -85,B 0,C 180,E1 -20850.815,E2 -20850.815} C_VEL
LIN {X 0,Y 218.298,Z 330.849,A -85,B 0,C 180,E1 -20851.781,E2 -20851.781} C_VEL
LIN {X 0,Y 217.447,Z 329.215,A -85,B 0,C 180,E1 -20852.175,E2 -20852.175} C_VEL
LIN {X 0,Y 215.168,Z 327.199,A -85,B 0,C 180,E1 -20853.127,E2 -20853.127} C_VEL
LIN {X 0,Y 213.954,Z 324.603,A -85,B 0,C 180,E1 -20853.742,E2 -20853.742} C_VEL
LIN {X 0,Y 213.797,Z 323.851,A -85,B 0,C 180,E1 -20853.918,E2 -20853.918} C_VEL
LIN {X 0,Y 213.793,Z 323.842,A -85,B 0,C 180,E1 -20858.802,E2 -20858.802} C_VEL
LIN {X 0,Y 213.932,Z 323.824,A -85,B 0,C 180,E1 -20862.803,E2 -20862.803} C_VEL
LIN {X 0,Y 213.941,Z 323.827,A -85,B 0,C 180,E1 -20866.706,E2 -20866.706} C_VEL
LIN {X 0,Y 214.124,Z 323.814,A -85,B 0,C 180,E1 -20870.555,E2 -20870.555} C_VEL
LIN {X 0,Y 214.077,Z 323.808,A -85,B 0,C 180,E1 -20874.348,E2 -20874.348} C_VEL
LIN {X 0,Y 214.431,Z 323.756,A -85,B 0,C 180,E1 -20878.122,E2 -20878.122} C_VEL
LIN {X 0,Y 214.538,Z 323.756,A -85,B 0,C 180,E1 -20880,E2 -20880} C_VEL
LIN {X 0,Y 214.433,Z 323.763,A -85,B 0,C 180,E1 -20881.879,E2 -20881.879} C_VEL
LIN {X 0,Y 214.216,Z 323.787,A -85,B 0,C 180,E1 -20887.541,E2 -20887.541} C_VEL
LIN {X 0,Y 214.033,Z 323.823,A -85,B 0,C 180,E1 -20891.363,E2 -20891.363} C_VEL
LIN {X 0,Y 213.922,Z 323.828,A -85,B 0,C 180,E1 -20895.238,E2 -20895.238} C_VEL
LIN {X 0,Y 213.828,Z 323.834,A -85,B 0,C 180,E1 -20899.189,E2 -20899.189} C_VEL
LIN {X 0,Y 213.837,Z 323.834,A -85,B 0,C 180,E1 -20903.229,E2 -20903.229} C_VEL
LIN {X 0,Y 213.819,Z 323.839,A -85,B 0,C 180,E1 -20907.452,E2 -20907.452} C_VEL
LIN {X 0,Y 213.77,Z 323.848,A -85,B 0,C 180,E1 -20911.738,E2 -20911.738} C_VEL
LIN {X 0,Y 213.762,Z 323.971,A -85,B 0,C 180,E1 -20916.468,E2 -20916.468} C_VEL
LIN {X 0,Y 215.075,Z 328.065,A -85,B 0,C 180,E1 -20919.584,E2 -20919.584} C_VEL
LIN {X 0,Y 216.33,Z 331.72,A -85,B 0,C 180,E1 -20922.1,E2 -20922.1} C_VEL
LIN {X 0,Y 217.357,Z 333.712,A -85,B 0,C 180,E1 -20922.582,E2 -20922.582} C_VEL
LIN {X 0,Y 220.033,Z 339.428,A -85,B 0,C 180,E1 -20923.817,E2 -20923.817} C_VEL
LIN {X 0,Y 226.609,Z 359.073,A -85,B 0,C 180,E1 -20926.858,E2 -20926.858} C_VEL
LIN {X 0,Y 232.76,Z 370.799,A -85,B 0,C 180,E1 -20929.096,E2 -20929.096} C_VEL
LIN {X 0,Y 238.273,Z 382.884,A -85,B 0,C 180,E1 -20930.99,E2 -20930.99} C_VEL
LIN {X 0,Y 240.042,Z 387.601,A -85,B 0,C 180,E1 -20931.601,E2 -20931.601} C_VEL
LIN {X 0,Y 241.184,Z 396.496,A -85,B 0,C 180,E1 -20932.228,E2 -20932.228} C_VEL
LIN {X 0,Y 238.493,Z 442.466,A -85,B 0,C 180,E1 -20933.571,E2 -20933.571} C_VEL
LIN {X 0,Y 236.792,Z 455.955,A -85,B 0,C 180,E1 -20934.248,E2 -20934.248} C_VEL
LIN {X 0,Y 234.524,Z 468.273,A -85,B 0,C 180,E1 -20935.166,E2 -20935.166} C_VEL
LIN {X 0,Y 231.539,Z 480.123,A -85,B 0,C 180,E1 -20936.365,E2 -20936.365} C_VEL
LIN {X 0,Y 228.173,Z 491.494,A -85,B 0,C 180,E1 -20937.909,E2 -20937.909} C_VEL
LIN {X 0,Y 224.681,Z 501.768,A -85,B 0,C 180,E1 -20939.713,E2 -20939.713} C_VEL
LIN {X 0,Y 221.405,Z 510.195,A -85,B 0,C 180,E1 -20941.57,E2 -20941.57} C_VEL
LIN {X 0,Y 217.396,Z 519.366,A -85,B 0,C 180,E1 -20944.127,E2 -20944.127} C_VEL
LIN {X 0,Y 213.951,Z 526.763,A -85,B 0,C 180,E1 -20946.788,E2 -20946.788} C_VEL
LIN {X 0,Y 211.254,Z 532.727,A -85,B 0,C 180,E1 -20949.558,E2 -20949.558} C_VEL
LIN {X 0,Y 208.835,Z 537.474,A -85,B 0,C 180,E1 -20952.373,E2 -20952.373} C_VEL
LIN {X 0,Y 206.899,Z 541.134,A -85,B 0,C 180,E1 -20955.244,E2 -20955.244} C_VEL
LIN {X 0,Y 205.626,Z 543.813,A -85,B 0,C 180,E1 -20958.169,E2 -20958.169} C_VEL
LIN {X 0,Y 204.64,Z 545.988,A -85,B 0,C 180,E1 -20962.107,E2 -20962.107} C_VEL
LIN {X 0,Y 204.406,Z 546.541,A -85,B 0,C 180,E1 -20966.06,E2 -20966.06} C_VEL
LIN {X 0,Y 204.466,Z 546.242,A -85,B 0,C 180,E1 -20968.033,E2 -20968.033} C_VEL
LIN {X 0,Y 204.597,Z 545.557,A -85,B 0,C 180,E1 -20970.003,E2 -20970.003} C_VEL
LIN {X 0,Y 204.509,Z 544.417,A -85,B 0,C 180,E1 -20971.972,E2 -20971.972} C_VEL
LIN {X 0,Y 204.437,Z 542.36,A -85,B 0,C 180,E1 -20974.476,E2 -20974.476} C_VEL
LIN {X 0,Y 204.68,Z 538.385,A -85,B 0,C 180,E1 -20977.897,E2 -20977.897} C_VEL
LIN {X 0,Y 205.163,Z 533.711,A -85,B 0,C 180,E1 -20980.863,E2 -20980.863} C_VEL
LIN {X 0,Y 206.258,Z 526.627,A -85,B 0,C 180,E1 -20984.305,E2 -20984.305} C_VEL
LIN {X 0,Y 207.766,Z 518.947,A -85,B 0,C 180,E1 -20987.219,E2 -20987.219} C_VEL
LIN {X 0,Y 209.337,Z 511.062,A -85,B 0,C 180,E1 -20989.62,E2 -20989.62} C_VEL
LIN {X 0,Y 211.364,Z 501.425,A -85,B 0,C 180,E1 -20991.97,E2 -20991.97} C_VEL
LIN {X 0,Y 213.116,Z 492.005,A -85,B 0,C 180,E1 -20993.83,E2 -20993.83} C_VEL
LIN {X 0,Y 214.637,Z 483.547,A -85,B 0,C 180,E1 -20995.196,E2 -20995.196} C_VEL
LIN {X 0,Y 216.575,Z 471.171,A -85,B 0,C 180,E1 -20996.763,E2 -20996.763} C_VEL
LIN {X 0,Y 218.23,Z 458.104,A -85,B 0,C 180,E1 -20997.971,E2 -20997.971} C_VEL
LIN {X 0,Y 219.413,Z 444.309,A -85,B 0,C 180,E1 -20998.811,E2 -20998.811} C_VEL
LIN {X 0,Y 220.549,Z 418.888,A -85,B 0,C 180,E1 -20999.664,E2 -20999.664} C_VEL
LIN {X 0,Y 221.485,Z 388.852,A -85,B 0,C 180,E1 -21000.621,E2 -21000.621} C_VEL
LIN {X 0,Y 217.912,Z 357.544,A -85,B 0,C 180,E1 -21002.193,E2 -21002.193} C_VEL
LIN {X 0,Y 212.619,Z 343.356,A -85,B 0,C 180,E1 -21003.434,E2 -21003.434} C_VEL
LIN {X 0,Y 208.756,Z 333.678,A -85,B 0,C 180,E1 -21004.377,E2 -21004.377} C_VEL
LIN {X 0,Y 206.695,Z 324.739,A -85,B 0,C 180,E1 -21008.551,E2 -21008.551} C_VEL
LIN {X 0,Y 206.63,Z 324.748,A -85,B 0,C 180,E1 -21012.867,E2 -21012.867} C_VEL
LIN {X 0,Y 206.63,Z 324.746,A -85,B 0,C 180,E1 -21017.136,E2 -21017.136} C_VEL
LIN {X 0,Y 206.695,Z 324.734,A -85,B 0,C 180,E1 -21021.451,E2 -21021.451} C_VEL
LIN {X 0,Y 206.707,Z 324.735,A -85,B 0,C 180,E1 -21024.69,E2 -21024.69} C_VEL
LIN {X 0,Y 206.732,Z 324.728,A -85,B 0,C 180,E1 -21029.34,E2 -21029.34} C_VEL
LIN {X 0,Y 206.74,Z 324.732,A -85,B 0,C 180,E1 -21033.773,E2 -21033.773} C_VEL
LIN {X 0,Y 206.743,Z 324.729,A -85,B 0,C 180,E1 -21038.041,E2 -21038.041} C_VEL
LIN {X 0,Y 206.83,Z 324.7,A -85,B 0,C 180,E1 -21042.192,E2 -21042.192} C_VEL
LIN {X 0,Y 206.888,Z 324.712,A -85,B 0,C 180,E1 -21046.243,E2 -21046.243} C_VEL
LIN {X 0,Y 207.087,Z 324.679,A -85,B 0,C 180,E1 -21050.23,E2 -21050.23} C_VEL
LIN {X 0,Y 207.055,Z 324.668,A -85,B 0,C 180,E1 -21054.155,E2 -21054.155} C_VEL
LIN {X 0,Y 207.386,Z 324.649,A -85,B 0,C 180,E1 -21058.058,E2 -21058.058} C_VEL
LIN {X 0,Y 207.519,Z 324.635,A -85,B 0,C 180,E1 -21060,E2 -21060} C_VEL
LIN {X 0,Y 207.388,Z 324.644,A -85,B 0,C 180,E1 -21061.942,E2 -21061.942} C_VEL
LIN {X 0,Y 207.144,Z 324.662,A -85,B 0,C 180,E1 -21067.799,E2 -21067.799} C_VEL
LIN {X 0,Y 206.927,Z 324.707,A -85,B 0,C 180,E1 -21071.758,E2 -21071.758} C_VEL
LIN {X 0,Y 206.837,Z 324.711,A -85,B 0,C 180,E1 -21075.773,E2 -21075.773} C_VEL
LIN {X 0,Y 206.754,Z 324.729,A -85,B 0,C 180,E1 -21079.872,E2 -21079.872} C_VEL
LIN {X 0,Y 206.754,Z 324.726,A -85,B 0,C 180,E1 -21084.073,E2 -21084.073} C_VEL
LIN {X 0,Y 206.751,Z 324.724,A -85,B 0,C 180,E1 -21088.417,E2 -21088.417} C_VEL
LIN {X 0,Y 206.709,Z 324.734,A -85,B 0,C 180,E1 -21092.955,E2 -21092.955} C_VEL
LIN {X 0,Y 206.686,Z 324.736,A -85,B 0,C 180,E1 -21097.738,E2 -21097.738} C_VEL
LIN {X 0,Y 206.648,Z 324.738,A -85,B 0,C 180,E1 -21101.561,E2 -21101.561} C_VEL
LIN {X 0,Y 206.637,Z 324.739,A -85,B 0,C 180,E1 -21105.58,E2 -21105.58} C_VEL
LIN {X 0,Y 206.665,Z 324.737,A -85,B 0,C 180,E1 -21109.747,E2 -21109.747} C_VEL
LIN {X 0,Y 206.704,Z 324.732,A -85,B 0,C 180,E1 -21114.687,E2 -21114.687} C_VEL
LIN {X 0,Y 206.711,Z 324.734,A -85,B 0,C 180,E1 -21119.334,E2 -21119.334} C_VEL
LIN {X 0,Y 206.738,Z 324.733,A -85,B 0,C 180,E1 -21123.77,E2 -21123.77} C_VEL
LIN {X 0,Y 206.782,Z 324.729,A -85,B 0,C 180,E1 -21128.043,E2 -21128.043} C_VEL
LIN {X 0,Y 206.818,Z 324.722,A -85,B 0,C 180,E1 -21130.6,E2 -21130.6} C_VEL
LIN {X 0,Y 207.875,Z 327.61,A -85,B 0,C 180,E1 -21130.874,E2 -21130.874} C_VEL
LIN {X 0,Y 214.867,Z 341.366,A -85,B 0,C 180,E1 -21132.406,E2 -21132.406} C_VEL
LIN {X 0,Y 218.802,Z 350.831,A -85,B 0,C 180,E1 -21133.282,E2 -21133.282} C_VEL
LIN {X 0,Y 222.313,Z 360.813,A -85,B 0,C 180,E1 -21134.086,E2 -21134.086} C_VEL
LIN {X 0,Y 220.712,Z 404.198,A -85,B 0,C 180,E1 -21135.439,E2 -21135.439} C_VEL
LIN {X 0,Y 219.695,Z 428.839,A -85,B 0,C 180,E1 -21136.268,E2 -21136.268} C_VEL
LIN {X 0,Y 218.671,Z 441.943,A -85,B 0,C 180,E1 -21137.055,E2 -21137.055} C_VEL
LIN {X 0,Y 217.381,Z 454.784,A -85,B 0,C 180,E1 -21138.221,E2 -21138.221} C_VEL
LIN {X 0,Y 215.646,Z 466.586,A -85,B 0,C 180,E1 -21139.671,E2 -21139.671} C_VEL
LIN {X 0,Y 213.879,Z 477.898,A -85,B 0,C 180,E1 -21141.494,E2 -21141.494} C_VEL
LIN {X 0,Y 212.063,Z 487.265,A -85,B 0,C 180,E1 -21143.374,E2 -21143.374} C_VEL
LIN {X 0,Y 210.207,Z 496.519,A -85,B 0,C 180,E1 -21145.683,E2 -21145.683} C_VEL
LIN {X 0,Y 208.284,Z 505.619,A -85,B 0,C 180,E1 -21148.547,E2 -21148.547} C_VEL
LIN {X 0,Y 206.782,Z 512.953,A -85,B 0,C 180,E1 -21151.458,E2 -21151.458} C_VEL
LIN {X 0,Y 205.873,Z 517.902,A -85,B 0,C 180,E1 -21153.912,E2 -21153.912} C_VEL
LIN {X 0,Y 205.204,Z 522.414,A -85,B 0,C 180,E1 -21156.682,E2 -21156.682} C_VEL
LIN {X 0,Y 204.518,Z 526.412,A -85,B 0,C 180,E1 -21159.89,E2 -21159.89} C_VEL
LIN {X 0,Y 204.246,Z 528.32,A -85,B 0,C 180,E1 -21161.912,E2 -21161.912} C_VEL
LIN {X 0,Y 204.187,Z 530.551,A -85,B 0,C 180,E1 -21165.477,E2 -21165.477} C_VEL
LIN {X 0,Y 204.329,Z 531.38,A -85,B 0,C 180,E1 -21168.029,E2 -21168.029} C_VEL
LIN {X 0,Y 204.637,Z 531.544,A -85,B 0,C 180,E1 -21170.083,E2 -21170.083} C_VEL
LIN {X 0,Y 205.163,Z 531.237,A -85,B 0,C 180,E1 -21172.347,E2 -21172.347} C_VEL
LIN {X 0,Y 206.595,Z 529.507,A -85,B 0,C 180,E1 -21176.243,E2 -21176.243} C_VEL
LIN {X 0,Y 207.71,Z 527.817,A -85,B 0,C 180,E1 -21178.391,E2 -21178.391} C_VEL
LIN {X 0,Y 209.627,Z 524.665,A -85,B 0,C 180,E1 -21181.305,E2 -21181.305} C_VEL
LIN {X 0,Y 212.093,Z 520.243,A -85,B 0,C 180,E1 -21184.282,E2 -21184.282} C_VEL
LIN {X 0,Y 215.091,Z 514.516,A -85,B 0,C 180,E1 -21187.187,E2 -21187.187} C_VEL
LIN {X 0,Y 218.59,Z 507.251,A -85,B 0,C 180,E1 -21190.014,E2 -21190.014} C_VEL
LIN {X 0,Y 222.521,Z 498.025,A -85,B 0,C 180,E1 -21192.765,E2 -21192.765} C_VEL
LIN {X 0,Y 226.228,Z 488.463,A -85,B 0,C 180,E1 -21194.969,E2 -21194.969} C_VEL
LIN {X 0,Y 229.786,Z 477.672,A -85,B 0,C 180,E1 -21196.9,E2 -21196.9} C_VEL
LIN {X 0,Y 232.692,Z 467.278,A -85,B 0,C 180,E1 -21198.359,E2 -21198.359} C_VEL
LIN {X 0,Y 235.261,Z 455.856,A -85,B 0,C 180,E1 -21199.615,E2 -21199.615} C_VEL
LIN {X 0,Y 237.489,Z 443.209,A -85,B 0,C 180,E1 -21200.622,E2 -21200.622} C_VEL
LIN {X 0,Y 239.055,Z 430.102,A -85,B 0,C 180,E1 -21201.323,E2 -21201.323} C_VEL
LIN {X 0,Y 240.74,Z 403.852,A -85,B 0,C 180,E1 -21202.109,E2 -21202.109} C_VEL
LIN {X 0,Y 242.022,Z 380.657,A -85,B 0,C 180,E1 -21202.768,E2 -21202.768} C_VEL
LIN {X 0,Y 235.979,Z 368.239,A -85,B 0,C 180,E1 -21204.734,E2 -21204.734} C_VEL
LIN {X 0,Y 230.186,Z 357.724,A -85,B 0,C 180,E1 -21206.728,E2 -21206.728} C_VEL
LIN {X 0,Y 224.061,Z 348.431,A -85,B 0,C 180,E1 -21208.964,E2 -21208.964} C_VEL
LIN {X 0,Y 220.245,Z 343.337,A -85,B 0,C 180,E1 -21210.441,E2 -21210.441} C_VEL
LIN {X 0,Y 217.354,Z 339.353,A -85,B 0,C 180,E1 -21211.647,E2 -21211.647} C_VEL
LIN {X 0,Y 214.964,Z 336.077,A -85,B 0,C 180,E1 -21212.695,E2 -21212.695} C_VEL
LIN {X 0,Y 213.629,Z 334.551,A -85,B 0,C 180,E1 -21213.285,E2 -21213.285} C_VEL
LIN {X 0,Y 211.497,Z 331.741,A -85,B 0,C 180,E1 -21214.284,E2 -21214.284} C_VEL
LIN {X 0,Y 210.697,Z 330.231,A -85,B 0,C 180,E1 -21214.699,E2 -21214.699} C_VEL
LIN {X 0,Y 208.245,Z 328.337,A -85,B 0,C 180,E1 -21215.846,E2 -21215.846} C_VEL
LIN {X 0,Y 206.97,Z 325.872,A -85,B 0,C 180,E1 -21216.565,E2 -21216.565} C_VEL
LIN {X 0,Y 206.756,Z 324.729,A -85,B 0,C 180,E1 -21216.816,E2 -21216.816} C_VEL
LIN {X 0,Y 206.861,Z 324.709,A -85,B 0,C 180,E1 -21222.196,E2 -21222.196} C_VEL
LIN {X 0,Y 206.883,Z 324.712,A -85,B 0,C 180,E1 -21226.244,E2 -21226.244} C_VEL
LIN {X 0,Y 207.068,Z 324.692,A -85,B 0,C 180,E1 -21230.23,E2 -21230.23} C_VEL
LIN {X 0,Y 207.039,Z 324.682,A -85,B 0,C 180,E1 -21234.156,E2 -21234.156} C_VEL
LIN {X 0,Y 207.367,Z 324.635,A -85,B 0,C 180,E1 -21238.058,E2 -21238.058} C_VEL
LIN {X 0,Y 207.503,Z 324.631,A -85,B 0,C 180,E1 -21240,E2 -21240} C_VEL
LIN {X 0,Y 207.369,Z 324.642,A -85,B 0,C 180,E1 -21241.943,E2 -21241.943} C_VEL
LIN {X 0,Y 207.156,Z 324.664,A -85,B 0,C 180,E1 -21247.8,E2 -21247.8} C_VEL
LIN {X 0,Y 206.97,Z 324.7,A -85,B 0,C 180,E1 -21251.756,E2 -21251.756} C_VEL
LIN {X 0,Y 206.856,Z 324.715,A -85,B 0,C 180,E1 -21255.772,E2 -21255.772} C_VEL
LIN {X 0,Y 206.773,Z 324.716,A -85,B 0,C 180,E1 -21259.871,E2 -21259.871} C_VEL
LIN {X 0,Y 206.754,Z 324.716,A -85,B 0,C 180,E1 -21264.074,E2 -21264.074} C_VEL
LIN {X 0,Y 206.735,Z 324.72,A -85,B 0,C 180,E1 -21268.421,E2 -21268.421} C_VEL
LIN {X 0,Y 206.701,Z 324.73,A -85,B 0,C 180,E1 -21272.958,E2 -21272.958} C_VEL
LIN {X 0,Y 206.73,Z 324.849,A -85,B 0,C 180,E1 -21273.974,E2 -21273.974} C_VEL
LIN {X 0,Y 208.604,Z 330.321,A -85,B 0,C 180,E1 -21278.557,E2 -21278.557} C_VEL
LIN {X 0,Y 208.948,Z 331.374,A -85,B 0,C 180,E1 -21279.184,E2 -21279.184} C_VEL
LIN {X 0,Y 211.826,Z 335.787,A -85,B 0,C 180,E1 -21280.627,E2 -21280.627} C_VEL
LIN {X 0,Y 213.518,Z 337.948,A -85,B 0,C 180,E1 -21281.408,E2 -21281.408} C_VEL
LIN {X 0,Y 216.584,Z 342.615,A -85,B 0,C 180,E1 -21282.799,E2 -21282.799} C_VEL
LIN {X 0,Y 221.398,Z 350.133,A -85,B 0,C 180,E1 -21284.823,E2 -21284.823} C_VEL
LIN {X 0,Y 226.357,Z 358.529,A -85,B 0,C 180,E1 -21286.758,E2 -21286.758} C_VEL
LIN {X 0,Y 226.609,Z 359.073,A -85,B 0,C 180,E1 -21286.858,E2 -21286.858} C_VEL
LIN {X 0,Y 228.78,Z 365.701,A -85,B 0,C 180,E1 -21287.79,E2 -21287.79} C_VEL
LIN {X 0,Y 232.712,Z 383.693,A -85,B 0,C 180,E1 -21289.656,E2 -21289.656} C_VEL
LIN {X 0,Y 233.838,Z 387.073,A -85,B 0,C 180,E1 -21290.089,E2 -21290.089} C_VEL
LIN {X 0,Y 235.18,Z 390.6,A -85,B 0,C 180,E1 -21290.574,E2 -21290.574} C_VEL
LIN {X 0,Y 236.031,Z 397.749,A -85,B 0,C 180,E1 -21291.085,E2 -21291.085} C_VEL
LIN {X 0,Y 233.291,Z 442.069,A -85,B 0,C 180,E1 -21292.388,E2 -21292.388} C_VEL
LIN {X 0,Y 231.487,Z 455.934,A -85,B 0,C 180,E1 -21293.094,E2 -21293.094} C_VEL
LIN {X 0,Y 229.026,Z 468.675,A -85,B 0,C 180,E1 -21294.068,E2 -21294.068} C_VEL
LIN {X 0,Y 225.72,Z 481.147,A -85,B 0,C 180,E1 -21295.377,E2 -21295.377} C_VEL
LIN {X 0,Y 222.235,Z 492.276,A -85,B 0,C 180,E1 -21296.944,E2 -21296.944} C_VEL
LIN {X 0,Y 218.617,Z 502.329,A -85,B 0,C 180,E1 -21298.78,E2 -21298.78} C_VEL
LIN {X 0,Y 214.505,Z 512.232,A -85,B 0,C 180,E1 -21301.105,E2 -21301.105} C_VEL
LIN {X 0,Y 210.377,Z 520.992,A -85,B 0,C 180,E1 -21303.731,E2 -21303.731} C_VEL
LIN {X 0,Y 206.913,Z 528.071,A -85,B 0,C 180,E1 -21306.504,E2 -21306.504} C_VEL
LIN {X 0,Y 204.601,Z 532.822,A -85,B 0,C 180,E1 -21308.862,E2 -21308.862} C_VEL
LIN {X 0,Y 202.08,Z 537.492,A -85,B 0,C 180,E1 -21311.763,E2 -21311.763} C_VEL
LIN {X 0,Y 200.027,Z 541.081,A -85,B 0,C 180,E1 -21314.725,E2 -21314.725} C_VEL
LIN {X 0,Y 198.646,Z 543.691,A -85,B 0,C 180,E1 -21317.747,E2 -21317.747} C_VEL
LIN {X 0,Y 198.031,Z 544.943,A -85,B 0,C 180,E1 -21319.782,E2 -21319.782} C_VEL
LIN {X 0,Y 197.59,Z 545.776,A -85,B 0,C 180,E1 -21321.824,E2 -21321.824} C_VEL
LIN {X 0,Y 197.326,Z 546.259,A -85,B 0,C 180,E1 -21325.918,E2 -21325.918} C_VEL
LIN {X 0,Y 197.366,Z 545.929,A -85,B 0,C 180,E1 -21327.962,E2 -21327.962} C_VEL
LIN {X 0,Y 197.51,Z 545.2,A -85,B 0,C 180,E1 -21330.003,E2 -21330.003} C_VEL
LIN {X 0,Y 197.407,Z 544.009,A -85,B 0,C 180,E1 -21332.043,E2 -21332.043} C_VEL
LIN {X 0,Y 197.346,Z 542.201,A -85,B 0,C 180,E1 -21334.317,E2 -21334.317} C_VEL
LIN {X 0,Y 197.502,Z 539.151,A -85,B 0,C 180,E1 -21337.157,E2 -21337.157} C_VEL
LIN {X 0,Y 197.938,Z 534.797,A -85,B 0,C 180,E1 -21340.229,E2 -21340.229} C_VEL
LIN {X 0,Y 198.734,Z 529.218,A -85,B 0,C 180,E1 -21343.292,E2 -21343.292} C_VEL
LIN {X 0,Y 200.155,Z 522.247,A -85,B 0,C 180,E1 -21346.317,E2 -21346.317} C_VEL
LIN {X 0,Y 201.695,Z 515.108,A -85,B 0,C 180,E1 -21348.806,E2 -21348.806} C_VEL
LIN {X 0,Y 203.001,Z 508.202,A -85,B 0,C 180,E1 -21350.81,E2 -21350.81} C_VEL
LIN {X 0,Y 204.907,Z 499.206,A -85,B 0,C 180,E1 -21352.966,E2 -21352.966} C_VEL
LIN {X 0,Y 206.961,Z 487.957,A -85,B 0,C 180,E1 -21355.12,E2 -21355.12} C_VEL
LIN {X 0,Y 209.052,Z 476.979,A -85,B 0,C 180,E1 -21356.724,E2 -21356.724} C_VEL
LIN {X 0,Y 210.86,Z 464.804,A -85,B 0,C 180,E1 -21358.088,E2 -21358.088} C_VEL
LIN {X 0,Y 212.26,Z 452.219,A -85,B 0,C 180,E1 -21359.101,E2 -21359.101} C_VEL
LIN {X 0,Y 213.266,Z 438.538,A -85,B 0,C 180,E1 -21359.788,E2 -21359.788} C_VEL
LIN {X 0,Y 215.05,Z 389.827,A -85,B 0,C 180,E1 -21361.374,E2 -21361.374} C_VEL
LIN {X 0,Y 211.687,Z 359.488,A -85,B 0,C 180,E1 -21362.952,E2 -21362.952} C_VEL
LIN {X 0,Y 204.329,Z 340.311,A -85,B 0,C 180,E1 -21364.766,E2 -21364.766} C_VEL
LIN {X 0,Y 201.451,Z 333.351,A -85,B 0,C 180,E1 -21365.526,E2 -21365.526} C_VEL
LIN {X 0,Y 199.615,Z 325.621,A -85,B 0,C 180,E1 -21369.33,E2 -21369.33} C_VEL
LIN {X 0,Y 199.58,Z 325.625,A -85,B 0,C 180,E1 -21372.311,E2 -21372.311} C_VEL
LIN {X 0,Y 199.585,Z 325.624,A -85,B 0,C 180,E1 -21375.229,E2 -21375.229} C_VEL
LIN {X 0,Y 199.586,Z 325.622,A -85,B 0,C 180,E1 -21378.006,E2 -21378.006} C_VEL
LIN {X 0,Y 199.618,Z 325.619,A -85,B 0,C 180,E1 -21380.769,E2 -21380.769} C_VEL
LIN {X 0,Y 199.621,Z 325.612,A -85,B 0,C 180,E1 -21385.715,E2 -21385.715} C_VEL
LIN {X 0,Y 199.709,Z 325.605,A -85,B 0,C 180,E1 -21388.138,E2 -21388.138} C_VEL
LIN {X 0,Y 199.695,Z 325.609,A -85,B 0,C 180,E1 -21392.772,E2 -21392.772} C_VEL
LIN {X 0,Y 199.721,Z 325.608,A -85,B 0,C 180,E1 -21397.227,E2 -21397.227} C_VEL
LIN {X 0,Y 199.756,Z 325.58,A -85,B 0,C 180,E1 -21401.802,E2 -21401.802} C_VEL
LIN {X 0,Y 199.825,Z 325.591,A -85,B 0,C 180,E1 -21405.747,E2 -21405.747} C_VEL
LIN {X 0,Y 200.032,Z 325.559,A -85,B 0,C 180,E1 -21409.882,E2 -21409.882} C_VEL
LIN {X 0,Y 200.017,Z 325.542,A -85,B 0,C 180,E1 -21413.949,E2 -21413.949} C_VEL
LIN {X 0,Y 200.325,Z 325.528,A -85,B 0,C 180,E1 -21417.989,E2 -21417.989} C_VEL
LIN {X 0,Y 200.484,Z 325.511,A -85,B 0,C 180,E1 -21420,E2 -21420} C_VEL
LIN {X 0,Y 200.029,Z 325.545,A -85,B 0,C 180,E1 -21424.029,E2 -21424.029} C_VEL
LIN {X 0,Y 200.094,Z 325.541,A -85,B 0,C 180,E1 -21428.076,E2 -21428.076} C_VEL
LIN {X 0,Y 199.876,Z 325.586,A -85,B 0,C 180,E1 -21432.179,E2 -21432.179} C_VEL
LIN {X 0,Y 199.774,Z 325.592,A -85,B 0,C 180,E1 -21436.346,E2 -21436.346} C_VEL
LIN {X 0,Y 199.679,Z 325.611,A -85,B 0,C 180,E1 -21440.607,E2 -21440.607} C_VEL
LIN {X 0,Y 199.672,Z 325.613,A -85,B 0,C 180,E1 -21444.984,E2 -21444.984} C_VEL
LIN {X 0,Y 199.682,Z 325.605,A -85,B 0,C 180,E1 -21449.521,E2 -21449.521} C_VEL
LIN {X 0,Y 199.684,Z 325.608,A -85,B 0,C 180,E1 -21452.356,E2 -21452.356} C_VEL
LIN {X 0,Y 199.63,Z 325.613,A -85,B 0,C 180,E1 -21456.761,E2 -21456.761} C_VEL
LIN {X 0,Y 199.615,Z 325.613,A -85,B 0,C 180,E1 -21459.326,E2 -21459.326} C_VEL
LIN {X 0,Y 199.58,Z 325.62,A -85,B 0,C 180,E1 -21462.308,E2 -21462.308} C_VEL
LIN {X 0,Y 199.583,Z 325.617,A -85,B 0,C 180,E1 -21465.226,E2 -21465.226} C_VEL
LIN {X 0,Y 199.583,Z 325.623,A -85,B 0,C 180,E1 -21468.003,E2 -21468.003} C_VEL
LIN {X 0,Y 199.615,Z 325.615,A -85,B 0,C 180,E1 -21470.766,E2 -21470.766} C_VEL
LIN {X 0,Y 199.617,Z 325.617,A -85,B 0,C 180,E1 -21475.711,E2 -21475.711} C_VEL
LIN {X 0,Y 199.697,Z 325.607,A -85,B 0,C 180,E1 -21478.133,E2 -21478.133} C_VEL
LIN {X 0,Y 199.691,Z 325.611,A -85,B 0,C 180,E1 -21482.769,E2 -21482.769} C_VEL
LIN {X 0,Y 199.754,Z 325.603,A -85,B 0,C 180,E1 -21487.228,E2 -21487.228} C_VEL
LIN {X 0,Y 199.741,Z 325.599,A -85,B 0,C 180,E1 -21489.509,E2 -21489.509} C_VEL
LIN {X 0,Y 200.75,Z 328.449,A -85,B 0,C 180,E1 -21489.794,E2 -21489.794} C_VEL
LIN {X 0,Y 207.479,Z 341.153,A -85,B 0,C 180,E1 -21491.343,E2 -21491.343} C_VEL
LIN {X 0,Y 212.211,Z 351.978,A -85,B 0,C 180,E1 -21492.439,E2 -21492.439} C_VEL
LIN {X 0,Y 215.95,Z 362.58,A -85,B 0,C 180,E1 -21493.341,E2 -21493.341} C_VEL
LIN {X 0,Y 213.216,Z 428.734,A -85,B 0,C 180,E1 -21495.502,E2 -21495.502} C_VEL
LIN {X 0,Y 212.124,Z 442.396,A -85,B 0,C 180,E1 -21496.343,E2 -21496.343} C_VEL
LIN {X 0,Y 210.847,Z 454.667,A -85,B 0,C 180,E1 -21497.484,E2 -21497.484} C_VEL
LIN {X 0,Y 208.904,Z 467.349,A -85,B 0,C 180,E1 -21499.089,E2 -21499.089} C_VEL
LIN {X 0,Y 207.09,Z 478.564,A -85,B 0,C 180,E1 -21500.967,E2 -21500.967} C_VEL
LIN {X 0,Y 205.125,Z 488.315,A -85,B 0,C 180,E1 -21503.011,E2 -21503.011} C_VEL
LIN {X 0,Y 203.089,Z 497.86,A -85,B 0,C 180,E1 -21505.531,E2 -21505.531} C_VEL
LIN {X 0,Y 201.127,Z 506.783,A -85,B 0,C 180,E1 -21508.495,E2 -21508.495} C_VEL
LIN {X 0,Y 199.644,Z 513.926,A -85,B 0,C 180,E1 -21511.51,E2 -21511.51} C_VEL
LIN {X 0,Y 198.485,Z 520.432,A -85,B 0,C 180,E1 -21515.075,E2 -21515.075} C_VEL
LIN {X 0,Y 197.734,Z 524.743,A -85,B 0,C 180,E1 -21518.17,E2 -21518.17} C_VEL
LIN {X 0,Y 197.345,Z 527.04,A -85,B 0,C 180,E1 -21520.254,E2 -21520.254} C_VEL
LIN {X 0,Y 197.127,Z 528.836,A -85,B 0,C 180,E1 -21522.348,E2 -21522.348} C_VEL
LIN {X 0,Y 197.113,Z 530.821,A -85,B 0,C 180,E1 -21525.704,E2 -21525.704} C_VEL
LIN {X 0,Y 197.312,Z 531.701,A -85,B 0,C 180,E1 -21528.694,E2 -21528.694} C_VEL
LIN {X 0,Y 198.164,Z 531.517,A -85,B 0,C 180,E1 -21532.765,E2 -21532.765} C_VEL
LIN {X 0,Y 198.961,Z 530.745,A -85,B 0,C 180,E1 -21535.076,E2 -21535.076} C_VEL
LIN {X 0,Y 200.898,Z 528.134,A -85,B 0,C 180,E1 -21539.006,E2 -21539.006} C_VEL
LIN {X 0,Y 203.246,Z 524.51,A -85,B 0,C 180,E1 -21542.406,E2 -21542.406} C_VEL
LIN {X 0,Y 205.948,Z 519.959,A -85,B 0,C 180,E1 -21545.455,E2 -21545.455} C_VEL
LIN {X 0,Y 209.169,Z 514.08,A -85,B 0,C 180,E1 -21548.428,E2 -21548.428} C_VEL
LIN {X 0,Y 212.911,Z 506.588,A -85,B 0,C 180,E1 -21551.309,E2 -21551.309} C_VEL
LIN {X 0,Y 216.364,Z 498.881,A -85,B 0,C 180,E1 -21553.645,E2 -21553.645} C_VEL
LIN {X 0,Y 220.197,Z 489.461,A -85,B 0,C 180,E1 -21555.896,E2 -21555.896} C_VEL
LIN {X 0,Y 223.907,Z 478.896,A -85,B 0,C 180,E1 -21557.858,E2 -21557.858} C_VEL
LIN {X 0,Y 227.241,Z 467.495,A -85,B 0,C 180,E1 -21559.498,E2 -21559.498} C_VEL
LIN {X 0,Y 230.051,Z 455.528,A -85,B 0,C 180,E1 -21560.818,E2 -21560.818} C_VEL
LIN {X 0,Y 232.254,Z 443.284,A -85,B 0,C 180,E1 -21561.791,E2 -21561.791} C_VEL
LIN {X 0,Y 233.893,Z 430.038,A -85,B 0,C 180,E1 -21562.5,E2 -21562.5} C_VEL
LIN {X 0,Y 236.133,Z 395.055,A -85,B 0,C 180,E1 -21563.541,E2 -21563.541} C_VEL
LIN {X 0,Y 236.727,Z 383.013,A -85,B 0,C 180,E1 -21563.912,E2 -21563.912} C_VEL
LIN {X 0,Y 231.614,Z 372.396,A -85,B 0,C 180,E1 -21565.669,E2 -21565.669} C_VEL
LIN {X 0,Y 225.92,Z 361.901,A -85,B 0,C 180,E1 -21567.744,E2 -21567.744} C_VEL
LIN {X 0,Y 219.997,Z 353.037,A -85,B 0,C 180,E1 -21570.016,E2 -21570.016} C_VEL
LIN {X 0,Y 216.738,Z 348.519,A -85,B 0,C 180,E1 -21571.361,E2 -21571.361} C_VEL
LIN {X 0,Y 214.34,Z 345.142,A -85,B 0,C 180,E1 -21572.41,E2 -21572.41} C_VEL
LIN {X 0,Y 211.16,Z 340.845,A -85,B 0,C 180,E1 -21573.872,E2 -21573.872} C_VEL
LIN {X 0,Y 208.637,Z 337.557,A -85,B 0,C 180,E1 -21575.099,E2 -21575.099} C_VEL
LIN {X 0,Y 207.682,Z 336.294,A -85,B 0,C 180,E1 -21575.583,E2 -21575.583} C_VEL
LIN {X 0,Y 205.115,Z 333.604,A -85,B 0,C 180,E1 -21576.893,E2 -21576.893} C_VEL
LIN {X 0,Y 203.734,Z 331.166,A -85,B 0,C 180,E1 -21577.701,E2 -21577.701} C_VEL
LIN {X 0,Y 201.197,Z 329.204,A -85,B 0,C 180,E1 -21579.087,E2 -21579.087} C_VEL
LIN {X 0,Y 199.984,Z 326.902,A -85,B 0,C 180,E1 -21579.896,E2 -21579.896} C_VEL
LIN {X 0,Y 199.734,Z 325.596,A -85,B 0,C 180,E1 -21580.204,E2 -21580.204} C_VEL
LIN {X 0,Y 199.792,Z 325.583,A -85,B 0,C 180,E1 -21583.656,E2 -21583.656} C_VEL
LIN {X 0,Y 199.862,Z 325.573,A -85,B 0,C 180,E1 -21587.82,E2 -21587.82} C_VEL
LIN {X 0,Y 200.065,Z 325.551,A -85,B 0,C 180,E1 -21591.923,E2 -21591.923} C_VEL
LIN {X 0,Y 200.306,Z 325.515,A -85,B 0,C 180,E1 -21597.99,E2 -21597.99} C_VEL
LIN {X 0,Y 200.467,Z 325.507,A -85,B 0,C 180,E1 -21600,E2 -21600} C_VEL
LIN {X 0,Y 200.017,Z 325.551,A -85,B 0,C 180,E1 -21604.03,E2 -21604.03} C_VEL
LIN {X 0,Y 200.1,Z 325.541,A -85,B 0,C 180,E1 -21608.077,E2 -21608.077} C_VEL
LIN {X 0,Y 199.902,Z 325.574,A -85,B 0,C 180,E1 -21612.178,E2 -21612.178} C_VEL
LIN {X 0,Y 199.794,Z 325.598,A -85,B 0,C 180,E1 -21616.345,E2 -21616.345} C_VEL
LIN {X 0,Y 199.69,Z 325.606,A -85,B 0,C 180,E1 -21620.607,E2 -21620.607} C_VEL
LIN {X 0,Y 199.664,Z 325.605,A -85,B 0,C 180,E1 -21624.986,E2 -21624.986} C_VEL
LIN {X 0,Y 199.666,Z 325.608,A -85,B 0,C 180,E1 -21629.524,E2 -21629.524} C_VEL
LIN {X 0,Y 199.67,Z 325.653,A -85,B 0,C 180,E1 -21630.983,E2 -21630.983} C_VEL
LIN {X 0,Y 201.328,Z 330.626,A -85,B 0,C 180,E1 -21635.622,E2 -21635.622} C_VEL
LIN {X 0,Y 204.65,Z 335.484,A -85,B 0,C 180,E1 -21637.558,E2 -21637.558} C_VEL
LIN {X 0,Y 206.278,Z 337.521,A -85,B 0,C 180,E1 -21638.425,E2 -21638.425} C_VEL
LIN {X 0,Y 210.03,Z 342.864,A -85,B 0,C 180,E1 -21640.337,E2 -21640.337} C_VEL
LIN {X 0,Y 213.733,Z 348.547,A -85,B 0,C 180,E1 -21642.098,E2 -21642.098} C_VEL
LIN {X 0,Y 218.183,Z 355.858,A -85,B 0,C 180,E1 -21644.071,E2 -21644.071} C_VEL
LIN {X 0,Y 222.718,Z 363.749,A -85,B 0,C 180,E1 -21645.926,E2 -21645.926} C_VEL
LIN {X 0,Y 228.572,Z 375.211,A -85,B 0,C 180,E1 -21648.177,E2 -21648.177} C_VEL
LIN {X 0,Y 233.752,Z 386.849,A -85,B 0,C 180,E1 -21650.058,E2 -21650.058} C_VEL
LIN {X 0,Y 233.838,Z 387.073,A -85,B 0,C 180,E1 -21650.089,E2 -21650.089} C_VEL
LIN {X 0,Y 234.61,Z 390.554,A -85,B 0,C 180,E1 -21650.432,E2 -21650.432} C_VEL
LIN {X 0,Y 234.571,Z 395.343,A -85,B 0,C 180,E1 -21650.629,E2 -21650.629} C_VEL
LIN {X 0,Y 233.335,Z 402.193,A -85,B 0,C 180,E1 -21650.623,E2 -21650.623} C_VEL
LIN {X 0,Y 230.307,Z 414.487,A -85,B 0,C 180,E1 -21650.409,E2 -21650.409} C_VEL
LIN {X 0,Y 229.793,Z 418.65,A -85,B 0,C 180,E1 -21650.464,E2 -21650.464} C_VEL
LIN {X 0,Y 228.071,Z 442.929,A -85,B 0,C 180,E1 -21651.207,E2 -21651.207} C_VEL
LIN {X 0,Y 226.289,Z 455.91,A -85,B 0,C 180,E1 -21651.887,E2 -21651.887} C_VEL
LIN {X 0,Y 223.874,Z 468.065,A -85,B 0,C 180,E1 -21652.825,E2 -21652.825} C_VEL
LIN {X 0,Y 220.426,Z 480.616,A -85,B 0,C 180,E1 -21654.14,E2 -21654.14} C_VEL
LIN {X 0,Y 216.822,Z 491.792,A -85,B 0,C 180,E1 -21655.727,E2 -21655.727} C_VEL
LIN {X 0,Y 213.051,Z 501.894,A -85,B 0,C 180,E1 -21657.589,E2 -21657.589} C_VEL
LIN {X 0,Y 209.063,Z 511.021,A -85,B 0,C 180,E1 -21659.722,E2 -21659.722} C_VEL
LIN {X 0,Y 204.739,Z 519.933,A -85,B 0,C 180,E1 -21662.396,E2 -21662.396} C_VEL
LIN {X 0,Y 200.976,Z 527.133,A -85,B 0,C 180,E1 -21665.192,E2 -21665.192} C_VEL
LIN {X 0,Y 197.985,Z 532.918,A -85,B 0,C 180,E1 -21668.12,E2 -21668.12} C_VEL
LIN {X 0,Y 195.351,Z 537.507,A -85,B 0,C 180,E1 -21671.111,E2 -21671.111} C_VEL
LIN {X 0,Y 193.152,Z 541.027,A -85,B 0,C 180,E1 -21674.167,E2 -21674.167} C_VEL
LIN {X 0,Y 191.685,Z 543.57,A -85,B 0,C 180,E1 -21677.295,E2 -21677.295} C_VEL
LIN {X 0,Y 191.024,Z 544.778,A -85,B 0,C 180,E1 -21679.403,E2 -21679.403} C_VEL
LIN {X 0,Y 190.281,Z 545.956,A -85,B 0,C 180,E1 -21683.642,E2 -21683.642} C_VEL
LIN {X 0,Y 190.236,Z 545.968,A -85,B 0,C 180,E1 -21685.937,E2 -21685.937} C_VEL
LIN {X 0,Y 190.269,Z 545.615,A -85,B 0,C 180,E1 -21687.886,E2 -21687.886} C_VEL
LIN {X 0,Y 190.426,Z 544.824,A -85,B 0,C 180,E1 -21690.003,E2 -21690.003} C_VEL
LIN {X 0,Y 190.307,Z 543.598,A -85,B 0,C 180,E1 -21692.12,E2 -21692.12} C_VEL
LIN {X 0,Y 190.269,Z 540.964,A -85,B 0,C 180,E1 -21695.302,E2 -21695.302} C_VEL
LIN {X 0,Y 190.568,Z 537.287,A -85,B 0,C 180,E1 -21698.486,E2 -21698.486} C_VEL
LIN {X 0,Y 191.168,Z 532.458,A -85,B 0,C 180,E1 -21701.669,E2 -21701.669} C_VEL
LIN {X 0,Y 192.196,Z 526.332,A -85,B 0,C 180,E1 -21704.834,E2 -21704.834} C_VEL
LIN {X 0,Y 193.821,Z 518.703,A -85,B 0,C 180,E1 -21707.955,E2 -21707.955} C_VEL
LIN {X 0,Y 195.396,Z 511.504,A -85,B 0,C 180,E1 -21710.328,E2 -21710.328} C_VEL
LIN {X 0,Y 197.703,Z 501.337,A -85,B 0,C 180,E1 -21713.022,E2 -21713.022} C_VEL
LIN {X 0,Y 199.795,Z 490.686,A -85,B 0,C 180,E1 -21715.249,E2 -21715.249} C_VEL
LIN {X 0,Y 202.043,Z 478.832,A -85,B 0,C 180,E1 -21717.168,E2 -21717.168} C_VEL
LIN {X 0,Y 204.07,Z 466.121,A -85,B 0,C 180,E1 -21718.688,E2 -21718.688} C_VEL
LIN {X 0,Y 205.703,Z 452.644,A -85,B 0,C 180,E1 -21719.84,E2 -21719.84} C_VEL
LIN {X 0,Y 206.721,Z 440.02,A -85,B 0,C 180,E1 -21720.523,E2 -21720.523} C_VEL
LIN {X 0,Y 208.622,Z 390.422,A -85,B 0,C 180,E1 -21722.193,E2 -21722.193} C_VEL
LIN {X 0,Y 205.542,Z 361.765,A -85,B 0,C 180,E1 -21723.739,E2 -21723.739} C_VEL
LIN {X 0,Y 198.477,Z 343.196,A -85,B 0,C 180,E1 -21725.575,E2 -21725.575} C_VEL
LIN {X 0,Y 194.146,Z 333.03,A -85,B 0,C 180,E1 -21726.771,E2 -21726.771} C_VEL
LIN {X 0,Y 192.529,Z 326.503,A -85,B 0,C 180,E1 -21730.185,E2 -21730.185} C_VEL
LIN {X 0,Y 192.497,Z 326.506,A -85,B 0,C 180,E1 -21733.926,E2 -21733.926} C_VEL
LIN {X 0,Y 192.52,Z 326.5,A -85,B 0,C 180,E1 -21738.921,E2 -21738.921} C_VEL
LIN {X 0,Y 192.594,Z 326.492,A -85,B 0,C 180,E1 -21743.403,E2 -21743.403} C_VEL
LIN {X 0,Y 192.619,Z 326.488,A -85,B 0,C 180,E1 -21747.059,E2 -21747.059} C_VEL
LIN {X 0,Y 192.674,Z 326.484,A -85,B 0,C 180,E1 -21751.693,E2 -21751.693} C_VEL
LIN {X 0,Y 192.693,Z 326.481,A -85,B 0,C 180,E1 -21756.346,E2 -21756.346} C_VEL
LIN {X 0,Y 192.704,Z 326.457,A -85,B 0,C 180,E1 -21761.491,E2 -21761.491} C_VEL
LIN {X 0,Y 192.749,Z 326.469,A -85,B 0,C 180,E1 -21765.212,E2 -21765.212} C_VEL
LIN {X 0,Y 192.954,Z 326.443,A -85,B 0,C 180,E1 -21769.567,E2 -21769.567} C_VEL
LIN {X 0,Y 192.98,Z 326.417,A -85,B 0,C 180,E1 -21773.727,E2 -21773.727} C_VEL
LIN {X 0,Y 193.267,Z 326.406,A -85,B 0,C 180,E1 -21777.916,E2 -21777.916} C_VEL
LIN {X 0,Y 193.448,Z 326.387,A -85,B 0,C 180,E1 -21780,E2 -21780} C_VEL
LIN {X 0,Y 192.975,Z 326.421,A -85,B 0,C 180,E1 -21784.177,E2 -21784.177} C_VEL
LIN {X 0,Y 193.042,Z 326.42,A -85,B 0,C 180,E1 -21788.373,E2 -21788.373} C_VEL
LIN {X 0,Y 192.802,Z 326.469,A -85,B 0,C 180,E1 -21792.633,E2 -21792.633} C_VEL
LIN {X 0,Y 192.727,Z 326.474,A -85,B 0,C 180,E1 -21796.961,E2 -21796.961} C_VEL
LIN {X 0,Y 192.616,Z 326.485,A -85,B 0,C 180,E1 -21801.399,E2 -21801.399} C_VEL
LIN {X 0,Y 192.655,Z 326.483,A -85,B 0,C 180,E1 -21804.211,E2 -21804.211} C_VEL
LIN {X 0,Y 192.657,Z 326.478,A -85,B 0,C 180,E1 -21808.89,E2 -21808.89} C_VEL
LIN {X 0,Y 192.606,Z 326.488,A -85,B 0,C 180,E1 -21813.184,E2 -21813.184} C_VEL
LIN {X 0,Y 192.558,Z 326.494,A -85,B 0,C 180,E1 -21818.35,E2 -21818.35} C_VEL
LIN {X 0,Y 192.497,Z 326.504,A -85,B 0,C 180,E1 -21823.094,E2 -21823.094} C_VEL
LIN {X 0,Y 192.495,Z 326.502,A -85,B 0,C 180,E1 -21826.903,E2 -21826.903} C_VEL
LIN {X 0,Y 192.556,Z 326.496,A -85,B 0,C 180,E1 -21831.646,E2 -21831.646} C_VEL
LIN {X 0,Y 192.601,Z 326.493,A -85,B 0,C 180,E1 -21836.811,E2 -21836.811} C_VEL
LIN {X 0,Y 192.665,Z 326.484,A -85,B 0,C 180,E1 -21841.689,E2 -21841.689} C_VEL
LIN {X 0,Y 192.701,Z 326.481,A -85,B 0,C 180,E1 -21847.481,E2 -21847.481} C_VEL
LIN {X 0,Y 192.68,Z 326.484,A -85,B 0,C 180,E1 -21848.324,E2 -21848.324} C_VEL
LIN {X 0,Y 193.72,Z 329.397,A -85,B 0,C 180,E1 -21848.644,E2 -21848.644} C_VEL
LIN {X 0,Y 198.372,Z 337.823,A -85,B 0,C 180,E1 -21849.791,E2 -21849.791} C_VEL
LIN {X 0,Y 204.549,Z 350.557,A -85,B 0,C 180,E1 -21851.277,E2 -21851.277} C_VEL
LIN {X 0,Y 209.012,Z 362.563,A -85,B 0,C 180,E1 -21852.396,E2 -21852.396} C_VEL
LIN {X 0,Y 209.581,Z 365.142,A -85,B 0,C 180,E1 -21852.575,E2 -21852.575} C_VEL
LIN {X 0,Y 206.788,Z 428.183,A -85,B 0,C 180,E1 -21854.662,E2 -21854.662} C_VEL
LIN {X 0,Y 205.734,Z 441.347,A -85,B 0,C 180,E1 -21855.468,E2 -21855.468} C_VEL
LIN {X 0,Y 204.353,Z 454.532,A -85,B 0,C 180,E1 -21856.7,E2 -21856.7} C_VEL
LIN {X 0,Y 202.446,Z 466.526,A -85,B 0,C 180,E1 -21858.229,E2 -21858.229} C_VEL
LIN {X 0,Y 200.588,Z 477.817,A -85,B 0,C 180,E1 -21860.14,E2 -21860.14} C_VEL
LIN {X 0,Y 198.447,Z 488.073,A -85,B 0,C 180,E1 -21862.314,E2 -21862.314} C_VEL
LIN {X 0,Y 196.357,Z 497.558,A -85,B 0,C 180,E1 -21864.863,E2 -21864.863} C_VEL
LIN {X 0,Y 194.276,Z 506.578,A -85,B 0,C 180,E1 -21867.924,E2 -21867.924} C_VEL
LIN {X 0,Y 192.688,Z 513.831,A -85,B 0,C 180,E1 -21871.042,E2 -21871.042} C_VEL
LIN {X 0,Y 191.579,Z 519.601,A -85,B 0,C 180,E1 -21874.204,E2 -21874.204} C_VEL
LIN {X 0,Y 190.805,Z 524.15,A -85,B 0,C 180,E1 -21877.403,E2 -21877.403} C_VEL
LIN {X 0,Y 190.197,Z 527.625,A -85,B 0,C 180,E1 -21880.644,E2 -21880.644} C_VEL
LIN {X 0,Y 189.997,Z 529.352,A -85,B 0,C 180,E1 -21882.82,E2 -21882.82} C_VEL
LIN {X 0,Y 190.018,Z 531.081,A -85,B 0,C 180,E1 -21885.923,E2 -21885.923} C_VEL
LIN {X 0,Y 190.326,Z 532.001,A -85,B 0,C 180,E1 -21889.407,E2 -21889.407} C_VEL
LIN {X 0,Y 191.229,Z 531.787,A -85,B 0,C 180,E1 -21893.25,E2 -21893.25} C_VEL
LIN {X 0,Y 192.217,Z 530.831,A -85,B 0,C 180,E1 -21896.021,E2 -21896.021} C_VEL
LIN {X 0,Y 194.111,Z 528.45,A -85,B 0,C 180,E1 -21899.665,E2 -21899.665} C_VEL
LIN {X 0,Y 196.945,Z 524.358,A -85,B 0,C 180,E1 -21903.577,E2 -21903.577} C_VEL
LIN {X 0,Y 199.891,Z 519.669,A -85,B 0,C 180,E1 -21906.702,E2 -21906.702} C_VEL
LIN {X 0,Y 203.345,Z 513.601,A -85,B 0,C 180,E1 -21909.742,E2 -21909.742} C_VEL
LIN {X 0,Y 207.346,Z 505.945,A -85,B 0,C 180,E1 -21912.675,E2 -21912.675} C_VEL
LIN {X 0,Y 210.883,Z 498.323,A -85,B 0,C 180,E1 -21914.975,E2 -21914.975} C_VEL
LIN {X 0,Y 215.09,Z 488.358,A -85,B 0,C 180,E1 -21917.318,E2 -21917.318} C_VEL
LIN {X 0,Y 218.97,Z 477.423,A -85,B 0,C 180,E1 -21919.306,E2 -21919.306} C_VEL
LIN {X 0,Y 222.326,Z 466.269,A -85,B 0,C 180,E1 -21920.869,E2 -21920.869} C_VEL
LIN {X 0,Y 224.926,Z 455.151,A -85,B 0,C 180,E1 -21922.083,E2 -21922.083} C_VEL
LIN {X 0,Y 227.353,Z 441.845,A -85,B 0,C 180,E1 -21923.111,E2 -21923.111} C_VEL
LIN {X 0,Y 228.964,Z 428.721,A -85,B 0,C 180,E1 -21923.782,E2 -21923.782} C_VEL
LIN {X 0,Y 231.626,Z 385.635,A -85,B 0,C 180,E1 -21925.071,E2 -21925.071} C_VEL
LIN {X 0,Y 226.583,Z 374.984,A -85,B 0,C 180,E1 -21926.927,E2 -21926.927} C_VEL
LIN {X 0,Y 221.722,Z 366.128,A -85,B 0,C 180,E1 -21928.799,E2 -21928.799} C_VEL
LIN {X 0,Y 216.361,Z 358.008,A -85,B 0,C 180,E1 -21930.974,E2 -21930.974} C_VEL
LIN {X 0,Y 211.253,Z 350.743,A -85,B 0,C 180,E1 -21933.251,E2 -21933.251} C_VEL
LIN {X 0,Y 208.22,Z 346.629,A -85,B 0,C 180,E1 -21934.71,E2 -21934.71} C_VEL
LIN {X 0,Y 205.017,Z 342.381,A -85,B 0,C 180,E1 -21936.358,E2 -21936.358} C_VEL
LIN {X 0,Y 202.438,Z 339.406,A -85,B 0,C 180,E1 -21937.752,E2 -21937.752} C_VEL
LIN {X 0,Y 201.208,Z 337.492,A -85,B 0,C 180,E1 -21938.485,E2 -21938.485} C_VEL
LIN {X 0,Y 198.694,Z 335.126,A -85,B 0,C 180,E1 -21939.962,E2 -21939.962} C_VEL
LIN {X 0,Y 197.191,Z 332.226,A -85,B 0,C 180,E1 -21941.022,E2 -21941.022} C_VEL
LIN {X 0,Y 194.485,Z 330.338,A -85,B 0,C 180,E1 -21942.791,E2 -21942.791} C_VEL
LIN {X 0,Y 193.032,Z 327.789,A -85,B 0,C 180,E1 -21943.95,E2 -21943.95} C_VEL
LIN {X 0,Y 192.743,Z 326.464,A -85,B 0,C 180,E1 -21944.333,E2 -21944.333} C_VEL
LIN {X 0,Y 192.933,Z 326.444,A -85,B 0,C 180,E1 -21949.567,E2 -21949.567} C_VEL
LIN {X 0,Y 192.963,Z 326.432,A -85,B 0,C 180,E1 -21953.728,E2 -21953.728} C_VEL
LIN {X 0,Y 193.248,Z 326.394,A -85,B 0,C 180,E1 -21957.916,E2 -21957.916} C_VEL
LIN {X 0,Y 193.431,Z 326.382,A -85,B 0,C 180,E1 -21960,E2 -21960} C_VEL
LIN {X 0,Y 192.963,Z 326.43,A -85,B 0,C 180,E1 -21964.178,E2 -21964.178} C_VEL
LIN {X 0,Y 193.05,Z 326.417,A -85,B 0,C 180,E1 -21968.374,E2 -21968.374} C_VEL
LIN {X 0,Y 192.841,Z 326.449,A -85,B 0,C 180,E1 -21972.631,E2 -21972.631} C_VEL
LIN {X 0,Y 192.747,Z 326.47,A -85,B 0,C 180,E1 -21976.96,E2 -21976.96} C_VEL
LIN {X 0,Y 192.627,Z 326.491,A -85,B 0,C 180,E1 -21981.399,E2 -21981.399} C_VEL
LIN {X 0,Y 192.654,Z 326.472,A -85,B 0,C 180,E1 -21984.227,E2 -21984.227} C_VEL
LIN {X 0,Y 192.643,Z 326.484,A -85,B 0,C 180,E1 -21987.425,E2 -21987.425} C_VEL
LIN {X 0,Y 193.866,Z 330.07,A -85,B 0,C 180,E1 -21991.332,E2 -21991.332} C_VEL
LIN {X 0,Y 196.452,Z 333.995,A -85,B 0,C 180,E1 -21993.234,E2 -21993.234} C_VEL
LIN {X 0,Y 199.383,Z 337.53,A -85,B 0,C 180,E1 -21995.126,E2 -21995.126} C_VEL
LIN {X 0,Y 202.438,Z 341.914,A -85,B 0,C 180,E1 -21996.96,E2 -21996.96} C_VEL
LIN {X 0,Y 203.887,Z 343.981,A -85,B 0,C 180,E1 -21997.776,E2 -21997.776} C_VEL
LIN {X 0,Y 207.847,Z 349.878,A -85,B 0,C 180,E1 -21999.877,E2 -21999.877} C_VEL
LIN {X 0,Y 211.777,Z 356.14,A -85,B 0,C 180,E1 -22001.804,E2 -22001.804} C_VEL
LIN {X 0,Y 215.338,Z 362.127,A -85,B 0,C 180,E1 -22003.434,E2 -22003.434} C_VEL
LIN {X 0,Y 219.769,Z 370.188,A -85,B 0,C 180,E1 -22005.333,E2 -22005.333} C_VEL
LIN {X 0,Y 224.719,Z 380.196,A -85,B 0,C 180,E1 -22007.326,E2 -22007.326} C_VEL
LIN {X 0,Y 229.491,Z 391.226,A -85,B 0,C 180,E1 -22009.16,E2 -22009.16} C_VEL
LIN {X 0,Y 230.459,Z 394.02,A -85,B 0,C 180,E1 -22009.538,E2 -22009.538} C_VEL
LIN {X 0,Y 230.963,Z 398.807,A -85,B 0,C 180,E1 -22009.881,E2 -22009.881} C_VEL
LIN {X 0,Y 229.793,Z 418.65,A -85,B 0,C 180,E1 -22010.464,E2 -22010.464} C_VEL
LIN {X 0,Y 228.964,Z 424.502,A -85,B 0,C 180,E1 -22010.508,E2 -22010.508} C_VEL
LIN {X 0,Y 223.428,Z 443.478,A -85,B 0,C 180,E1 -22010.066,E2 -22010.066} C_VEL
LIN {X 0,Y 222.275,Z 449.228,A -85,B 0,C 180,E1 -22010.238,E2 -22010.238} C_VEL
LIN {X 0,Y 220.081,Z 461.804,A -85,B 0,C 180,E1 -22011.05,E2 -22011.05} C_VEL
LIN {X 0,Y 217.261,Z 473.324,A -85,B 0,C 180,E1 -22012.08,E2 -22012.08} C_VEL
LIN {X 0,Y 213.793,Z 484.607,A -85,B 0,C 180,E1 -22013.433,E2 -22013.433} C_VEL
LIN {X 0,Y 209.647,Z 496.083,A -85,B 0,C 180,E1 -22015.261,E2 -22015.261} C_VEL
LIN {X 0,Y 205.355,Z 506.271,A -85,B 0,C 180,E1 -22017.387,E2 -22017.387} C_VEL
LIN {X 0,Y 200.7,Z 516.063,A -85,B 0,C 180,E1 -22020.07,E2 -22020.07} C_VEL
LIN {X 0,Y 196.392,Z 523.97,A -85,B 0,C 180,E1 -22022.857,E2 -22022.857} C_VEL
LIN {X 0,Y 193.473,Z 529.226,A -85,B 0,C 180,E1 -22025.25,E2 -22025.25} C_VEL
LIN {X 0,Y 190.399,Z 534.618,A -85,B 0,C 180,E1 -22028.342,E2 -22028.342} C_VEL
LIN {X 0,Y 187.766,Z 538.761,A -85,B 0,C 180,E1 -22031.452,E2 -22031.452} C_VEL
LIN {X 0,Y 185.679,Z 541.877,A -85,B 0,C 180,E1 -22034.639,E2 -22034.639} C_VEL
LIN {X 0,Y 184.745,Z 543.451,A -85,B 0,C 180,E1 -22036.809,E2 -22036.809} C_VEL
LIN {X 0,Y 184.035,Z 544.596,A -85,B 0,C 180,E1 -22038.996,E2 -22038.996} C_VEL
LIN {X 0,Y 183.213,Z 545.706,A -85,B 0,C 180,E1 -22043.395,E2 -22043.395} C_VEL
LIN {X 0,Y 183.153,Z 545.641,A -85,B 0,C 180,E1 -22046.105,E2 -22046.105} C_VEL
LIN {X 0,Y 183.342,Z 544.447,A -85,B 0,C 180,E1 -22050.003,E2 -22050.003} C_VEL
LIN {X 0,Y 183.163,Z 541.889,A -85,B 0,C 180,E1 -22053.943,E2 -22053.943} C_VEL
LIN {X 0,Y 183.378,Z 538.119,A -85,B 0,C 180,E1 -22057.712,E2 -22057.712} C_VEL
LIN {X 0,Y 183.907,Z 533.614,A -85,B 0,C 180,E1 -22061.019,E2 -22061.019} C_VEL
LIN {X 0,Y 185.074,Z 526.749,A -85,B 0,C 180,E1 -22064.855,E2 -22064.855} C_VEL
LIN {X 0,Y 186.713,Z 519.263,A -85,B 0,C 180,E1 -22068.095,E2 -22068.095} C_VEL
